PLC2_RANGE_7_1 3325.07 BOOL  ; IN RANGE 7 COUNTER 1
PLC2_RANGE_7_2 3326.07 BOOL  ; IN RANGE 7 COUNTER 2
PLC2_RANGE_8_1 3325.08 BOOL  ; IN RANGE 8 COUNTER 1
PLC2_RANGE_8_2 3326.08 BOOL  ; IN RANGE 8 COUNTER 2
PLC2_RANGE_9_1 3325.09 BOOL  ; IN RANGE 9 COUNTER 1
PLC2_RANGE_9_2 3326.09 BOOL  ; IN RANGE 9 COUNTER 2
PLC3_RANGE_12_1 3325.12 BOOL  ; IN RANGE 12 COUNTER 1
PLC3_RANGE_14_1 3325.14 BOOL  ; IN RANGE 14 COUNTER 1
PRESET_INC_HAG W225.05 BOOL  ; PRESET INCLINOMETER AT HAGENBUCH SYSTEM
PULSE_ENTANCE_GATE_RIGHT W161.00 BOOL  ; PULSE TO OPEN AND CLOSE ENTRANCE GATE RIGHT
PULSE_ENTRANCE_GATE_LEFT W161.01 BOOL  ; PULSE TO OPEN AND CLOSE ENTRANCE GATE LEFT
PULSE_EXIT_GATE W166.00 BOOL  ; PULSE TO OPEN AND CLOSE EXIT GATE
R2_COUNTER4_H 364 INT  ; VALUE COUNTER 4 HIGH WORD
R2_COUNTER_4_L 363 INT  ; VALUE COUNTER 4 LOW WORD
R2_COUNTER_5 369 INT  ; ANALOGE SPANNING KUNSTMATIGE HORIZON
RAMP_DN_X1 D7014 REAL  ; BEGINNING OF RAMP AREA
RAMP_DN_X2 D7016 REAL  ; END OF RAMP AREA
RAMP_DN_Y1 D7010 REAL  ; MAX SPEED AT THE END OF RAMP
RAMP_DN_Y2 D7012 REAL  ; MAX SPEED AT THE BEGINNING OF RAMP
RAMP_FACTOR D182 CHANNEL  ; RAMP FACTOR FOR ARM MOTION
RAMP_UP_X1 D7004 REAL  ; BEGINNING OF RAMP AREA
RAMP_UP_X2 D7006 REAL  ; END OF RAMP AREA
RAMP_UP_Y1 D7000 REAL  ; MAX SPEED AT THE END OF RAMP
RAMP_UP_Y2 D7002 REAL  ; MAX SPEED AT THE BEGINNING OF RAMP
RESULT_A_DN D7074 REAL  ; RESULT A DOWN
RESULT_A_UP D7054 REAL  ; RESULT A UP
RESULT_A_X_DN D7072 REAL  ; RESULT A X DOWN
RESULT_A_X_UP D7052 REAL  ; RESULT A X UP
RESULT_A_Y_DN D7070 REAL  ; RESULT A Y DOWN
RESULT_A_Y_UP D7050 REAL  ; RESULT A Y UP
RESULT_B1_DN D7076 REAL  ; RESULT B1 DOWN
RESULT_B1_UP D7056 REAL  ; RESULT B1 UP
RESULT_B2_DN D7082 REAL  ; RESULT B2 DOWN
RESULT_B2_UP D7062 REAL  ; RESULT B2 UP
RESULT_B_DN D7078 REAL  ; RESULT B DOWN
RESULT_B_UP D7058 REAL  ; RESULT B UP
RESULT_COUNTER_01 2022 INT  ; PULS GETAL ENCODER 1
RESULT_COUNTER_02 2024 INT  ; PULS GETAL ENCODER 2
RESULT_POSITION_VAR_A_DN D7080 REAL  ; RESULT POSITION * VAR A DOWN
RESULT_POSITION_VAR_A_UP D7060 REAL  ; RESULT POSITION * VAR A UP
RES_14_03 14.03 BOOL
RES_14_04 14.04 BOOL
RES_14_05 14.05 BOOL
RES_14_06 14.06 BOOL
RES_14_07 14.07 BOOL
RES_14_08 14.08 BOOL
RES_14_09 14.09 BOOL
RES_14_10 14.10 BOOL
RES_14_11 14.11 BOOL
RES_14_12 14.12 BOOL
RES_14_13 14.13 BOOL
RES_14_14 14.14 BOOL
RES_14_15 14.15 BOOL
STOP_ARM_GOING_UP 3338.00 BOOL  ; STOP ARM GOING UP (LINK BIT TO PLC 1)
TIMER_1 T0001 BOOL L  ; TEST 1
TIMER_2 T0002 BOOL L  ; TEST 2
TIMER_ENC1_FAULT 0150 NUMBER  ; TIMER ENCODER 1 FAUT
TIMER_ENC2_FAULT 0151 NUMBER  ; TIMER ENCODER 2 FAULT
TIMER_PULSE_GATE 0165 NUMBER  ; TIMER FOR OPEN AND CLOSE PULSE EXIT GATE
TIMER_PULSE_GATE_LEFT 0161 NUMBER  ; TIMER FOR OPEN AND CLOSE PULSE ENTRANCE GATE LEFT
TIMER_PULSE_GATE_RIGHT 0160 NUMBER  ; TIMER FOR OPEN AND CLOSE PULSE ENTRANCE GATE RIGHT
TIMER_RESET_BIT 0301 NUMBER  ; TIMER RESET STOP ARM GOING UP BIT
TIMER_STOP_ARM_UP 0300 NUMBER  ; TIMER STOP ARM UP
T_ALARM_1_0161_SET T0021 BOOL
T_ALARM_1_0162_SET T0022 BOOL
T_ALARM_1_0164_SET T0023 BOOL
T_ALARM_1_1191 0320 NUMBER  ; Timer Alarm 1191
T_ALARM_1_1192 0321 NUMBER  ; Timer Alarm 1192
T_ALARM_1_1347 T0205 BOOL
T_ALARM_1_1347_SET 205 NUMBER
T_ALARM_1_1350 T0206 BOOL
T_ALARM_1_1350_SET 206 NUMBER
T_ALARM_1_1453 T0223 BOOL  ; ALARM 1-1453 SIGNAL STATUS VALVE 47 NOT OK
T_ALARM_1_1456 0223 NUMBER  ; ALARM 1-1456 INFO LINK HAGENBUCH (FIBRE OPTIK) NOT AVAILABLE
T_ALARM_1_1457 0224 NUMBER  ; ALARM 1-1457 INFO LINK HAGENBUCH TOO MANY ERRORS
T_ALARM_1_1458 0225 NUMBER  ; ALARM 1-1458 INCLINOMETER TO STABILIZE THE ISLAND NOT OK
T_ALARM_1_1459 0226 NUMBER  ; ALARM 1-1459 STABLIZATION ANGLE ERROR (NORMAL BEFORE TILT SWITCH ERROR)
T_ALARM_1_1460 0227 NUMBER  ; ALARM 1-1460 STABLIZATION PUMP OUT OF ZERO POSITION (MUST BE ZERO POSITION WHEN INLAND IN HOME POSITION)
T_ALARM_1_1461 0228 NUMBER  ; ALARM 1-1461 STABLIZATION PUMP NOT OK
T_ALARM_1_1462_OFF 0231 NUMBER  ; ALARM 1-1462 HARDWARE WATCHDOG FROM HAGENBUCH MISSING TIMER OFF
T_ALARM_1_1462_ON 0230 NUMBER  ; ALARM 1-1462 HARDWARE WATCHDOG FROM HAGENBUCH MISSING TIMER ON
T_ARM_HYDRAULIC_ON 0240 NUMBER  ; TIMER ARM HYDRAULIC ON
T_EILAND_BOVEN T0115 BOOL  ; EILAND TIJD BOVEN
T_Hydr_Main_Pump_Arm_On 0194 NUMBER  ; Hydraulic main pump arm on delay timer
T_ING_L_DICHT T0163 BOOL  ; Max Tijd Sluit Linker Poortjes Oever
T_ING_L_DICHT_SET 161 NUMBER  ; MAX TIJD SLUITEN INGANGS POORT LINKS
T_ING_L_OPEN T0162 BOOL  ; Max Tijd Open Linker Poortjes Oever
T_ING_L_OPEN_SET 160 NUMBER  ; MAX TIJD OPENE INGANG LINKS
T_ING_R_DICHT T0161 BOOL  ; Max Tijd Sluit Rechter Poortjes Oever
T_ING_R_DICHT_SET 163 NUMBER  ; MAX TIJD OPEPEN INGANGS POORTEN RECHTS
T_ING_R_OPEN T0160 BOOL  ; Max Tijd Open Rechter Poortjes Oever
T_ING_R_OPEN_SET 162 NUMBER  ; MAX TIJD OPEPEN INGANGS POORT RECTS
T_ISLAND_HYDRAULIC_ON 0241 NUMBER  ; TIMER ISLAND HYDRAULIC ON
T_Input_0_00 500 NUMBER
T_MS_11Q08_not_OK 0195 NUMBER  ; Hydraulic main pump arm MS 11Q08 not OK
T_MS_11Q10_not_OK 0196 NUMBER  ; Hydraulic main pump arm MS 11Q10 not OK
T_MS_11Q12_not_OK 0197 NUMBER  ; Hydraulic main pump arm MS 11Q12 not OK
T_Open_Uitgangs_poortjes T0165 BOOL  ; Maximale tijd Open Uitgangs Poortjes
T_PRESET_INC_HAGENBUCH 0311 NUMBER  ; PRESET INCLINOMETER HAGENBUCH
T_RESET_HAGENBUCH 0310 NUMBER  ; TIMER RESET ERROR HAGENBUCH SYSTEM
T_SNELHEID 145 NUMBER  ; SNELHEIDS METING ARM
T_SNELHEID_ACT T0145 BOOL  ; TIMER TBV ARM SNELEHEID
T_STUURDRUK_SET_GROND 170 NUMBER  ; DELAY STUURDRUK AANWEZIG
T_STUUR_DRUK T0170 BOOL  ; DELAY STUURDRUK MOET AANWEZIG ZIJN
T_STUUR_DRUK_EIL T0220 BOOL  ; STUURDRUK AANWEZIG EILAND
T_SUURDRUK_EILAND_SET 220 NUMBER  ; DELAY STUUR DRUK AANWEZIG
T_UITG_DICHT T0169 BOOL  ; MAX TIJD UITGANGS POORT SLUITEN
T_UITG_DICHT_SET 169 NUMBER  ; MAX TIJD SLUITEN UITGANGS POORT
T_UITG_OPEN T0165 BOOL  ; MAX TIJD OPENEN UITGANGS POORT
T_UITG_OPEN_SET 165 NUMBER  ; MAX TIJD OPENEN UITGANGS POORTEN
T_Watchdog_Pulse_Check_Plc_2_H T0020 BOOL
T_Watchdog_Pulse_Check_Plc_2_L T0024 BOOL
T_Watchdog_Pulse_Check_Plc_2_Set_H 20 NUMBER
T_Watchdog_Pulse_Check_Plc_2_Set_L 25 NUMBER
T_eilandpoort_set 164 NUMBER  ; delay eilandpoort melding
T_eilandpoortje_act T0164 BOOL  ; delay eiland poort melding
Test_Speed D7500 REAL
U2_72K10 60.03 BOOL  ; ENABLE LINKSOM FREQ.REGELAAR MOTOREN ROTATIE
U2_72K12 60.04 BOOL  ; VRIJGEVEN MOTORREM 1,2,3 EN 4 ROTATIE EILAND
U2_72K14 60.05 BOOL  ; BYPASS ISLAND STABILISATION PUMP
U2_72K16 60.06 BOOL  ; VRIJGAVE POORTJES EILAND
U2_72K18 60.07 BOOL  ; BYPASS ISLAND STABILISATION CYLINDER
U2_72K6 60.01 BOOL L  ; VOEDING FREQ.REGELAAR MOTOREN ROTATIE
U2_72K8 60.02 BOOL  ; ENABLE RECHTSOM FREQ.REGELAAR MOTOREN ROTATIE
U2_73K6 61.02 BOOL  ; HOOFDMOTOR HYDRAULIEK EILAND
U2_73K8 61.03 BOOL  ; VRIJGAVE POORTJES EILAND
U2_73Q4 61.01 BOOL  ; STUURPOMP HYDRAULIEK EILAND
U2_CNT4_COUNT_READ 64.06 BOOL  ; READ COUNTER VALUE
U2_CNT4_COUNT_SET 64.02 BOOL  ; COUNTING SET BIT
U2_CNT4_MODE_1 64.11 BOOL  ; DIFF PHASE 1x
U2_CNT4_MODE_2 64.10 BOOL  ; DIFF PHASE 1x
U2_CNT4_MODE_3 64.12 BOOL  ; RESET MODE
U2_CNT4_MODE_4 64.13 BOOL  ; RESET MODE
U2_CNT4_MODE_5 64.14 BOOL  ; RESET MODE
U2_CNT4_MODE_7 64.03 BOOL  ; DATA MODE 0=BCD 1=HEX
U2_CNT4_RESET 64.07 BOOL  ; INTERNAL RESET
U2_NOOD_PCL1A 60.00 BOOL L  ; NOODSTOP CIRCUIT REMOTE I/O PLC1
U2_NOOD_PCL1B 61.00 BOOL  ; NOODSTOP CIRCUIT REMOTE I/O PLC1
U2_RES_01 61.07 BOOL
U2_SHOWLIGHT_01 61.05 BOOL  ; SHOWLIGHT 01
U2_SHOWLIGHT_02 61.06 BOOL  ; SHOWLIGHT 02
UPS_fault H121.03 BOOL  ; UPS in storing of batterij bedrijf
U_44SH12 13.14 BOOL  ; Ingangs poortjes links oever
U_44SH14 13.15 BOOL  ; Ingangs Poortjes Rechts Oever
U_55K4 8.01 BOOL  ; WATCH DOG PLC 1 (UITGANG DEFECT!!!)
U_85K10 8.04 BOOL  ; ONTGRENDELEN TOURNIQUET LINKS
U_85K12 8.05 BOOL  ; ONTGRENDELEN TOURNIQUET RECHTS
U_85K4 8.07 BOOL  ; Tijdelijke uitgang tbv watchdog
U_85K4_1 7.00 BOOL  ; WATCH DOG PLC 2 NIEUW
U_85Y14 8.06 BOOL  ; POORTJE RECHTS INGANG OPENEN (OEVER)
U_85Y6 8.02 BOOL  ; ARM OMHOOG KLEP 1
U_85Y8 8.03 BOOL  ; ARM OMLAAG KLEP 1
U_86Y10 9.04 BOOL  ; ARM OMLAAG KLEP 3
U_86Y4 9.01 BOOL  ; ARM OMHOOG KLEP 2
U_86Y6 9.02 BOOL  ; ARM OMLAAG KLEP 2
U_86Y8 9.03 BOOL  ; ARM OMHOOG KLEP 3
U_87K8 10.03 BOOL  ; START HOOFDMOTOR HYDRAULIEK UNIT ARM
U_87Q10 10.04 BOOL  ; START STUURPOMP HYDRAULIEK UNIT ARM
U_87Q12 10.05 BOOL  ; START SMEERTOESTEL HYDRAULIEK UNIT ARM
U_87Q14 10.06 BOOL  ; START OLIEREINIGING HYDRAULIEK UNIT ARM
U_87Q6 10.02 BOOL  ; START OLIEKOELER HYDRAULIEK UNIT ARM
U_87Y2 10.00 BOOL  ; POORTJE UITGANG OPENEN (OEVER)
U_87Y4 10.01 BOOL  ; POORTJE UITGANG SLUITEN (OEVER)
U_88Z12 11.05 BOOL  ; ALGEMEEN ALARM ZOEMER
U_91H10 13.04 BOOL  ; ALGEMEEN ALARM
U_91H12 13.05 BOOL  ; KLAAR VOOR SHOW
U_91H14 13.06 BOOL  ; TOURNIQUET LINKS ONTGRENDELD
U_91H16 13.07 BOOL  ; TOURNIQUET RECHTS ONTGRENDELD
U_91H18 13.08 BOOL  ; ARM (EILAND) OMHOOG
U_91H2 13.00 BOOL  ; STUURSPANNING IN
U_91H4 13.01 BOOL  ; HAND BEDRIJF
U_91H6 13.02 BOOL  ; AUTOMATISCH BEDRIJF
U_91H8 13.03 BOOL  ; POMPEN IN BEDRIJF
U_92H12 13.13 BOOL  ; Reset Noodstop
U_92H2 13.09 BOOL  ; ARM (EILAND) OMLAAG
U_92H4 13.10 BOOL  ; EILAND ROTATIE LINKSOM
U_92H6 13.11 BOOL  ; EILAND ROTATIE RECHTSOM
U_92H8 13.12 BOOL  ; Service mode
U_ANA_ARM 2041 CHANNEL  ; ANALOOG _UIT_CHAN1 TBV ARM BESTURING
U_Analog_Uit_Ch2 66 CHANNEL  ; ANALOG OUTPUT ARM POSITION IN DEGREE
U_Analog_Uit_Ch4 68 CHANNEL  ; ANALOG OUTPUT ARM SPEED IN DEGREE/MINUTE
U_ENAB_ANA_CHAN1 2040.00 BOOL  ; CHAN 1 ENABLE
U_ENTRACE_GATE_RIGHT 14.00 BOOL  ; ENTRANCE GATE RIGHT
U_ENTRANCE_GATE_LEFT 14.01 BOOL  ; ENTRANCE GATE LEFT
U_EXIT_GATE 14.02 BOOL  ; EXIT GATE
U_HAG_BIT_10 61.04 BOOL  ; HAGENBUCH TILT SENSOREN OK
U_HAG_PRESET 9.05 BOOL  ; HAGENBUCH PRESET INCLINOMETER
U_HAG_RESET 9.06 BOOL  ; HAGENBUCH ALARM RESET
U_Ingangs_Poortje_Links_Oever 12.04 BOOL
U_Ingangs_Poortje_Rechts_Oever 12.00 BOOL
U_NS_PLC1A 8.00 BOOL  ; NOODSTOP CIRCUIT PLC 1
U_NS_PLC1B 9.00 BOOL  ; NOODSTOP CIRCUIT PLC 1
U_Open_Ingangs_Poortje_2_Links_Oever 12.05 BOOL
U_Open_Ingangs_Poortje_2_Rechts_Oever 12.01 BOOL  ; Open Ingangs Poortje 2 Rechter zijde Oever
U_Open_Uitgangs_Poortje_2_Oever 12.09 BOOL
U_RES_10_07 10.07 BOOL  ; RESERVE
U_Res_noodstop 9.07 BOOL  ; Mogelijk om noodstop te resetten
U_Sluit_Ingangs_Poortje_1_Links_Oever 12.06 BOOL
U_Sluit_Ingangs_Poortje_1_Rechts_Oever 12.02 BOOL  ; Sluit Poortje 1 Rechter zijde Oever
U_Sluit_Ingangs_Poortje_2_Links_Oever 12.07 BOOL
U_Sluit_Ingangs_Poortje_2_Rechts_Oever 12.03 BOOL  ; Sluit Poortje 2 Rechter zijde Oever
U_Sluit_Uitgangs_Poortje_1_Oever 12.10 BOOL
U_Sluit_Uitgangs_Poortje_2_Oever 12.11 BOOL
U_Uitgangs_Poortje_Oever 12.08 BOOL
W_ING_PRT_EIL_GESL W210.05 BOOL  ; Ingangs Poortjes Eiland Gesloten Plc 1 & 2 & 3
W_RANGE0_CNT1 W125.00 BOOL  ; ARM IN RANGE 0
W_RANGE0_CNT2 W126.00 BOOL  ; ARM IN RANGE 0
W_RANGE0_PLC1 3036.00 BOOL  ; ARM IN RANGE 0
W_RANGE0_PLC2 3336.00 BOOL  ; ARM IN RANGE 0
W_RANGE10_CNT1 W125.10 BOOL  ; ARM IN RANGE 10
W_RANGE10_CNT2 W126.10 BOOL  ; ARM IN RANGE 10
W_RANGE10_PLC1 3036.10 BOOL  ; ARM IN RANGE 10
W_RANGE10_PLC2 3336.10 BOOL  ; ARM IN RANGE 10
W_RANGE11_CNT1 W125.11 BOOL  ; ARM IN RANGE 11
W_RANGE11_CNT2 W126.11 BOOL  ; ARM IN RANGE 11
W_RANGE11_PLC1 3036.11 BOOL  ; ARM IN RANGE 11
W_RANGE11_PLC2 3336.11 BOOL  ; ARM IN RANGE 11
W_RANGE12_CNT1 W125.12 BOOL  ; ARM IN RANGE 12
W_RANGE12_CNT2 W126.12 BOOL  ; ARM IN RANGE 12
W_RANGE12_PLC1 3036.12 BOOL  ; ARM IN RANGE 12
W_RANGE12_PLC2 3336.12 BOOL  ; ARM IN RANGE 12
W_RANGE13_CNT1 W125.13 BOOL  ; ARM IN RANGE 13
W_RANGE13_CNT2 W126.13 BOOL  ; ARM IN RANGE 13
W_RANGE13_PLC1 3036.13 BOOL  ; ARM IN RANGE 13
W_RANGE13_PLC2 3336.13 BOOL  ; ARM IN RANGE 13
W_RANGE14_CNT1 W125.14 BOOL  ; ARM IN RANGE 14
W_RANGE14_CNT2 W126.14 BOOL  ; ARM IN RANGE 14
W_RANGE14_PLC1 3036.14 BOOL  ; ARM IN RANGE 14
W_RANGE14_PLC2 3336.14 BOOL  ; ARM IN RANGE 14
W_RANGE15_CNT1 W125.15 BOOL  ; ARM IN RANGE 15
W_RANGE15_CNT2 W126.15 BOOL  ; ARM IN RANGE 15
W_RANGE15_PLC1 3036.15 BOOL  ; ARM IN RANGE 15
W_RANGE15_PLC2 3336.15 BOOL  ; ARM IN RANGE 15
W_RANGE1_CNT1 W125.01 BOOL  ; ARM IN RANGE 1
W_RANGE1_CNT2 W126.01 BOOL  ; ARM IN RANGE 1
W_RANGE1_PLC1 3036.01 BOOL  ; ARM IN RANGE 1
W_RANGE1_PLC2 3336.01 BOOL  ; ARM IN RANGE 1
W_RANGE2_CNT1 W125.02 BOOL  ; ARM IN RANGE 2
W_RANGE2_CNT2 W126.02 BOOL  ; ARM IN RANGE 2
W_RANGE2_PLC1 3036.02 BOOL  ; ARM IN RANGE 2
W_RANGE2_PLC2 3336.02 BOOL  ; ARM IN RANGE 2
W_RANGE3_CNT1 W125.03 BOOL  ; ARM IN RANGE 3
W_RANGE3_CNT2 W126.03 BOOL  ; ARM IN RANGE 3
W_RANGE3_PLC1 3036.03 BOOL  ; ARM IN RANGE 3
W_RANGE3_PLC2 3336.03 BOOL  ; ARM IN RANGE 3
W_RANGE4_CNT1 W125.04 BOOL  ; ARM IN RANGE 4
W_RANGE4_CNT2 W126.04 BOOL  ; ARM IN RANGE 4
W_RANGE4_PLC1 3036.04 BOOL  ; ARM IN RANGE 4
W_RANGE4_PLC2 3336.04 BOOL  ; ARM IN RANGE 4
W_RANGE5_CNT1 W125.05 BOOL  ; ARM IN RANGE 5
W_RANGE5_CNT2 W126.05 BOOL  ; ARM IN RANGE 5
W_RANGE5_PLC1 3036.05 BOOL  ; ARM IN RANGE 5
W_RANGE5_PLC2 3336.05 BOOL  ; ARM IN RANGE 5
W_RANGE6_CNT1 W125.06 BOOL  ; ARM IN RANGE 6
W_RANGE6_CNT2 W126.06 BOOL  ; ARM IN RANGE 6
W_RANGE6_PLC1 3036.06 BOOL  ; ARM IN RANGE 6
W_RANGE6_PLC2 3336.06 BOOL  ; ARM IN RANGE 6
W_RANGE7_CNT1 W125.07 BOOL  ; ARM IN RANGE 7
W_RANGE7_CNT2 W126.07 BOOL  ; ARM IN RANGE 7
W_RANGE7_PLC1 3036.07 BOOL  ; ARM IN RANGE 7
W_RANGE7_PLC2 3336.07 BOOL  ; ARM IN RANGE 7
W_RANGE8_CNT1 W125.08 BOOL  ; ARM IN RANGE 8
W_RANGE8_CNT2 W126.08 BOOL  ; ARM IN RANGE 8
W_RANGE8_PLC1 3036.08 BOOL  ; ARM IN RANGE 8
W_RANGE8_PLC2 3336.08 BOOL  ; ARM IN RANGE 8
W_RANGE9_CNT1 W125.09 BOOL  ; ARM IN RANGE 9
W_RANGE9_CNT2 W126.09 BOOL  ; ARM IN RANGE 9
W_RANGE9_PLC1 3036.09 BOOL  ; ARM IN RANGE 9
W_RANGE9_PLC2 3336.09 BOOL  ; ARM IN RANGE 9
com1_Eiland_Home 3024.02 BOOL  ; Het Eiland Is geheel Links- of Rechtsom Gedraaid
t_diff_arm T0175 BOOL  ; verschil soll-ist arm
t_diff_soll_arm 175 NUMBER  ; diff soll ist verschil arm
t_eiland_boven 0115 NUMBER  ; eiland boven tijd

## Program ALGEMEEN (cyclic task 0)
Local symbols
M_ALARM_1_0000 H100.00 BOOL  ; Alarm 1 - 0000 Er is minstens 1 Alarm in de File Main (Alarmen 1 - 0000 t/m 1 -  0031)
M_ALARM_1_0032 H102.00 BOOL  ; Alarm 1 - 0032 Er is minstens 1 Alarm in de Controllink (Alarmen 1 - 0032 t/m 1 -  0063)
M_ALARM_1_0096 H106.00 BOOL  ; Alarm 1 - 0096 Er is minstens 1 Alarm in de Data-Opslag (Alarmen 1 - 0096 t/m 1 -  0127)
M_ALARM_1_0128 H108.00 BOOL  ; Alarm 1-0128 Er is minstens 1 alarm in de I/O Controle afhandeling
M_Alarm_H100_H108 W36.00 BOOL
M_Alarm_H110_H118 W36.01 BOOL
M_Alarm_H120_H128 W36.02 BOOL
M_Alarm_H130_H138 W36.03 BOOL
M_Alarm_H140_H148 W36.04 BOOL
M_Alarm_H150_H158 W36.05 BOOL
M_Alarm_H160_H168 W36.06 BOOL
M_Alarm_H170_H178 W36.07 BOOL
M_Alarm_H180_H188 W36.08 BOOL
M_Alarm_H190_H198 W36.09 BOOL
U_WCD_1 11.06 BOOL
U_WCD_2 11.07 BOOL
U_WCD_5 61.07 BOOL

### Section Main

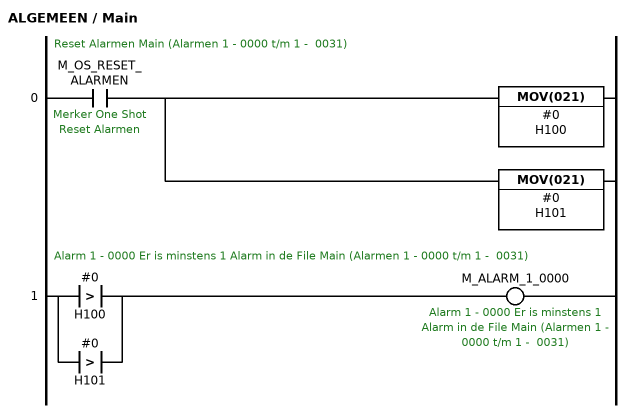
; rung 0: Reset Alarmen Main (Alarmen 1 - 0000 t/m 1 -  0031)
LD M_OS_RESET_ALARMEN  ; Merker One Shot Reset Alarmen
MOV(021) #0 H100
MOV(021) #0 H101
; rung 1: Alarm 1 - 0000 Er is minstens 1 Alarm in de File Main (Alarmen 1 - 0000 t/m 1 -  0031)
LD>(320) #0 H100
OR>(320) #0 H101
OUT M_ALARM_1_0000  ; Alarm 1 - 0000 Er is minstens 1 Alarm in de File Main (Alarmen 1 - 0000 t/m 1 -  0031)

### Section Control_Link

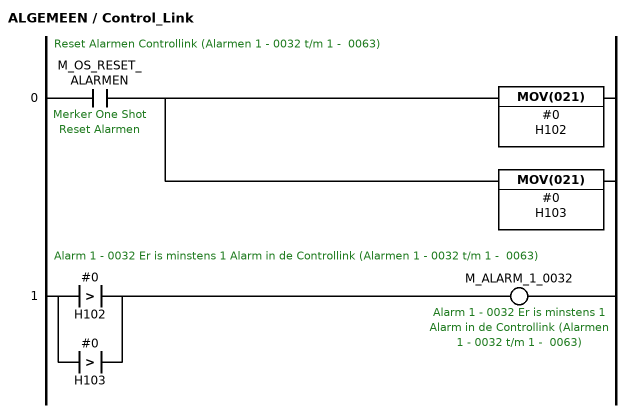
; rung 0: Reset Alarmen Controllink (Alarmen 1 - 0032 t/m 1 -  0063)
LD M_OS_RESET_ALARMEN  ; Merker One Shot Reset Alarmen
MOV(021) #0 H102
MOV(021) #0 H103
; rung 1: Alarm 1 - 0032 Er is minstens 1 Alarm in de Controllink (Alarmen 1 - 0032 t/m 1 -  0063)
LD>(320) #0 H102
OR>(320) #0 H103
OUT M_ALARM_1_0032  ; Alarm 1 - 0032 Er is minstens 1 Alarm in de Controllink (Alarmen 1 - 0032 t/m 1 -  0063)

### Section Device_net

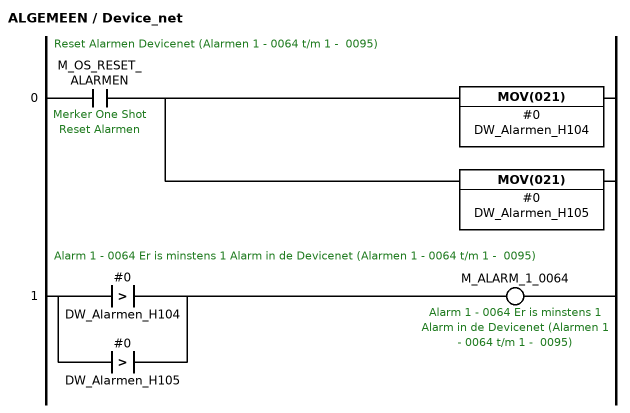
; rung 0: Reset Alarmen Devicenet (Alarmen 1 - 0064 t/m 1 -  0095)
LD M_OS_RESET_ALARMEN  ; Merker One Shot Reset Alarmen
MOV(021) #0 DW_Alarmen_H104
MOV(021) #0 DW_Alarmen_H105
; rung 1: Alarm 1 - 0064 Er is minstens 1 Alarm in de Devicenet (Alarmen 1 - 0064 t/m 1 -  0095)
LD>(320) #0 DW_Alarmen_H104
OR>(320) #0 DW_Alarmen_H105
OUT M_ALARM_1_0064  ; Alarm 1 - 0064 Er is minstens 1 Alarm in de Devicenet (Alarmen 1 - 0064 t/m 1 -  0095)

### Section Data_Opslag

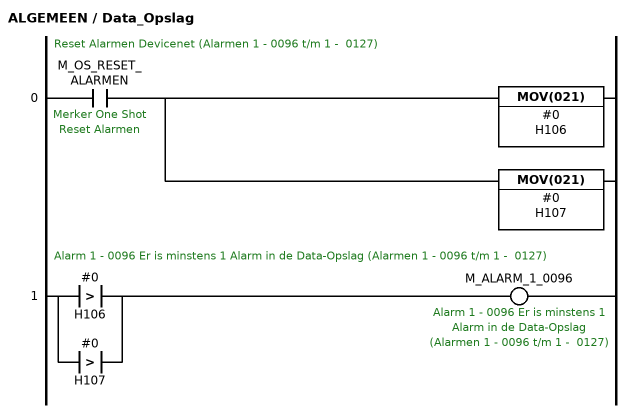
; rung 0: Reset Alarmen Devicenet (Alarmen 1 - 0096 t/m 1 -  0127)
LD M_OS_RESET_ALARMEN  ; Merker One Shot Reset Alarmen
MOV(021) #0 H106
MOV(021) #0 H107
; rung 1: Alarm 1 - 0096 Er is minstens 1 Alarm in de Data-Opslag (Alarmen 1 - 0096 t/m 1 -  0127)
LD>(320) #0 H106
OR>(320) #0 H107
OUT M_ALARM_1_0096  ; Alarm 1 - 0096 Er is minstens 1 Alarm in de Data-Opslag (Alarmen 1 - 0096 t/m 1 -  0127)

### Section I_O_Controle

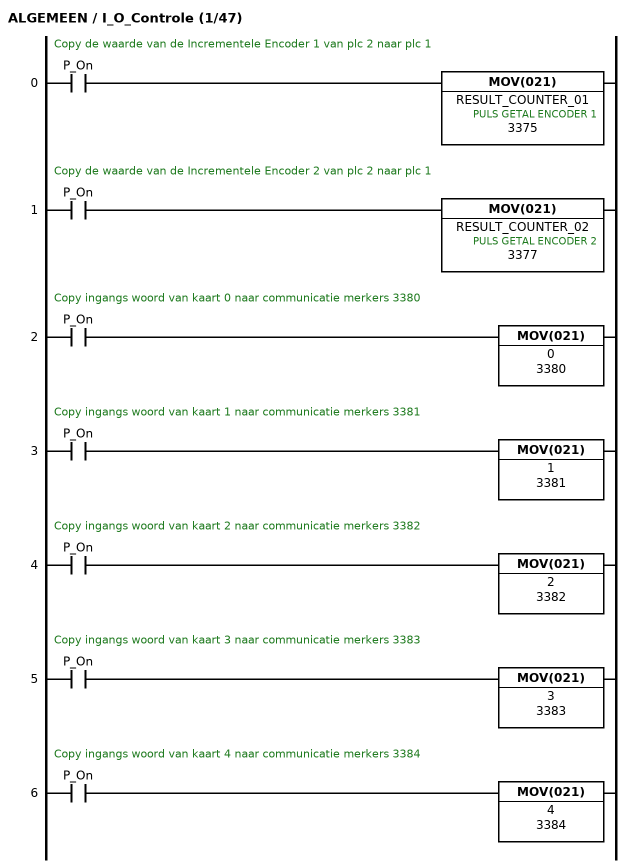
; rung 0: Copy de waarde van de Incrementele Encoder 1 van plc 2 naar plc 1
LD P_On
MOV(021) RESULT_COUNTER_01 3375  ; PULS GETAL ENCODER 1
; rung 1: Copy de waarde van de Incrementele Encoder 2 van plc 2 naar plc 1
LD P_On
MOV(021) RESULT_COUNTER_02 3377  ; PULS GETAL ENCODER 2
; rung 2: Copy ingangs woord van kaart 0 naar communicatie merkers 3380
LD P_On
MOV(021) 0 3380
; rung 3: Copy ingangs woord van kaart 1 naar communicatie merkers 3381
LD P_On
MOV(021) 1 3381
; rung 4: Copy ingangs woord van kaart 2 naar communicatie merkers 3382
LD P_On
MOV(021) 2 3382
; rung 5: Copy ingangs woord van kaart 3 naar communicatie merkers 3383
LD P_On
MOV(021) 3 3383
; rung 6: Copy ingangs woord van kaart 4 naar communicatie merkers 3384
LD P_On
MOV(021) 4 3384

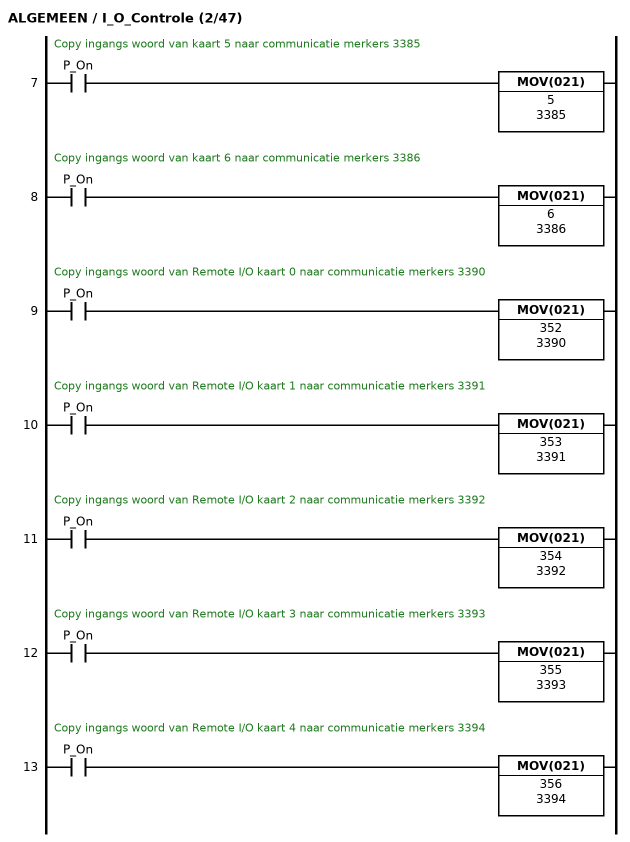
; rung 7: Copy ingangs woord van kaart 5 naar communicatie merkers 3385
LD P_On
MOV(021) 5 3385
; rung 8: Copy ingangs woord van kaart 6 naar communicatie merkers 3386
LD P_On
MOV(021) 6 3386
; rung 9: Copy ingangs woord van Remote I/O kaart 0 naar communicatie merkers 3390
LD P_On
MOV(021) 352 3390
; rung 10: Copy ingangs woord van Remote I/O kaart 1 naar communicatie merkers 3391
LD P_On
MOV(021) 353 3391
; rung 11: Copy ingangs woord van Remote I/O kaart 2 naar communicatie merkers 3392
LD P_On
MOV(021) 354 3392
; rung 12: Copy ingangs woord van Remote I/O kaart 3 naar communicatie merkers 3393
LD P_On
MOV(021) 355 3393
; rung 13: Copy ingangs woord van Remote I/O kaart 4 naar communicatie merkers 3394
LD P_On
MOV(021) 356 3394

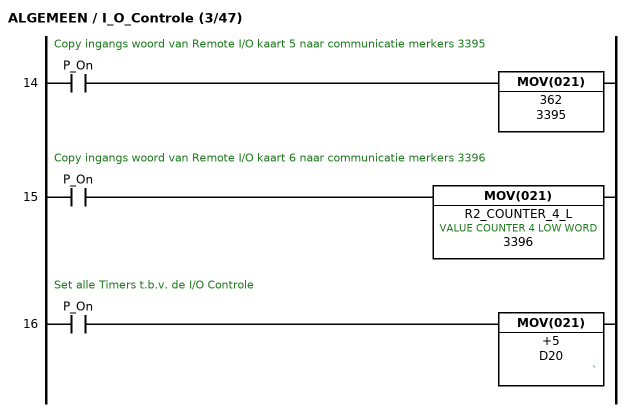
; rung 14: Copy ingangs woord van Remote I/O kaart 5 naar communicatie merkers 3395
LD P_On
MOV(021) 362 3395
; rung 15: Copy ingangs woord van Remote I/O kaart 6 naar communicatie merkers 3396
LD P_On
MOV(021) R2_COUNTER_4_L 3396  ; VALUE COUNTER 4 LOW WORD
; rung 16: Set alle Timers t.b.v. de I/O Controle
LD P_On
MOV(021) +5 D20  ; `

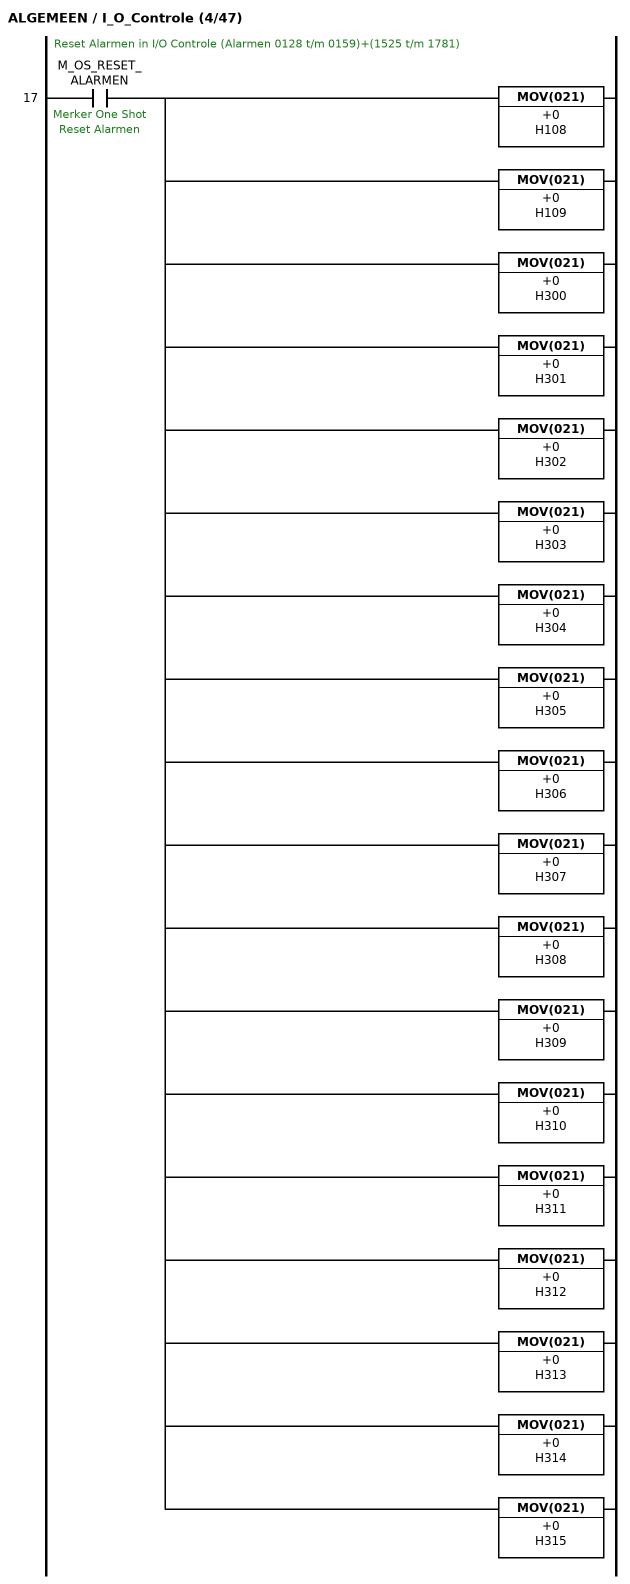
; rung 17: Reset Alarmen in I/O Controle (Alarmen 0128 t/m 0159)+(1525 t/m 1781)
LD M_OS_RESET_ALARMEN  ; Merker One Shot Reset Alarmen
MOV(021) +0 H108
MOV(021) +0 H109
MOV(021) +0 H300
MOV(021) +0 H301
MOV(021) +0 H302
MOV(021) +0 H303
MOV(021) +0 H304
MOV(021) +0 H305
MOV(021) +0 H306
MOV(021) +0 H307
MOV(021) +0 H308
MOV(021) +0 H309
MOV(021) +0 H310
MOV(021) +0 H311
MOV(021) +0 H312
MOV(021) +0 H313
MOV(021) +0 H314
MOV(021) +0 H315

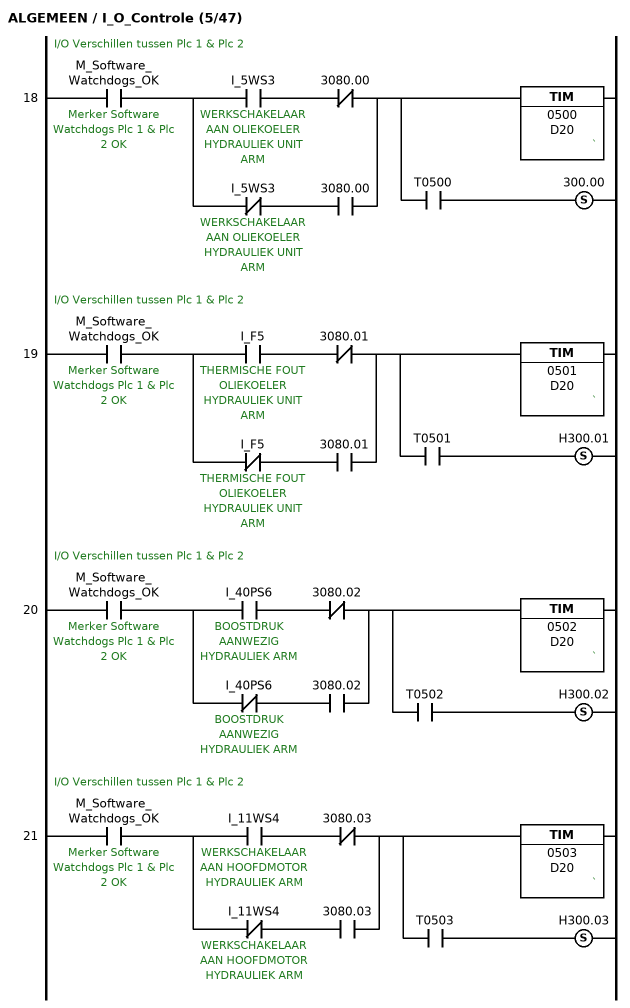
; rung 18: I/O Verschillen tussen Plc 1 & Plc 2
LD M_Software_Watchdogs_OK  ; Merker Software Watchdogs Plc 1 & Plc 2 OK
LD I_5WS3  ; WERKSCHAKELAAR AAN OLIEKOELER HYDRAULIEK UNIT ARM
ANDNOT 3080.00
LDNOT I_5WS3  ; WERKSCHAKELAAR AAN OLIEKOELER HYDRAULIEK UNIT ARM
AND 3080.00
ORLD
ANDLD
TIM 0500 D20  ; `
AND T0500
SET 300.00
; rung 19: I/O Verschillen tussen Plc 1 & Plc 2
LD M_Software_Watchdogs_OK  ; Merker Software Watchdogs Plc 1 & Plc 2 OK
LD I_F5  ; THERMISCHE FOUT OLIEKOELER HYDRAULIEK UNIT ARM
ANDNOT 3080.01
LDNOT I_F5  ; THERMISCHE FOUT OLIEKOELER HYDRAULIEK UNIT ARM
AND 3080.01
ORLD
ANDLD
TIM 0501 D20  ; `
AND T0501
SET H300.01
; rung 20: I/O Verschillen tussen Plc 1 & Plc 2
LD M_Software_Watchdogs_OK  ; Merker Software Watchdogs Plc 1 & Plc 2 OK
LD I_40PS6  ; BOOSTDRUK AANWEZIG HYDRAULIEK ARM
ANDNOT 3080.02
LDNOT I_40PS6  ; BOOSTDRUK AANWEZIG HYDRAULIEK ARM
AND 3080.02
ORLD
ANDLD
TIM 0502 D20  ; `
AND T0502
SET H300.02
; rung 21: I/O Verschillen tussen Plc 1 & Plc 2
LD M_Software_Watchdogs_OK  ; Merker Software Watchdogs Plc 1 & Plc 2 OK
LD I_11WS4  ; WERKSCHAKELAAR AAN HOOFDMOTOR HYDRAULIEK ARM
ANDNOT 3080.03
LDNOT I_11WS4  ; WERKSCHAKELAAR AAN HOOFDMOTOR HYDRAULIEK ARM
AND 3080.03
ORLD
ANDLD
TIM 0503 D20  ; `
AND T0503
SET H300.03

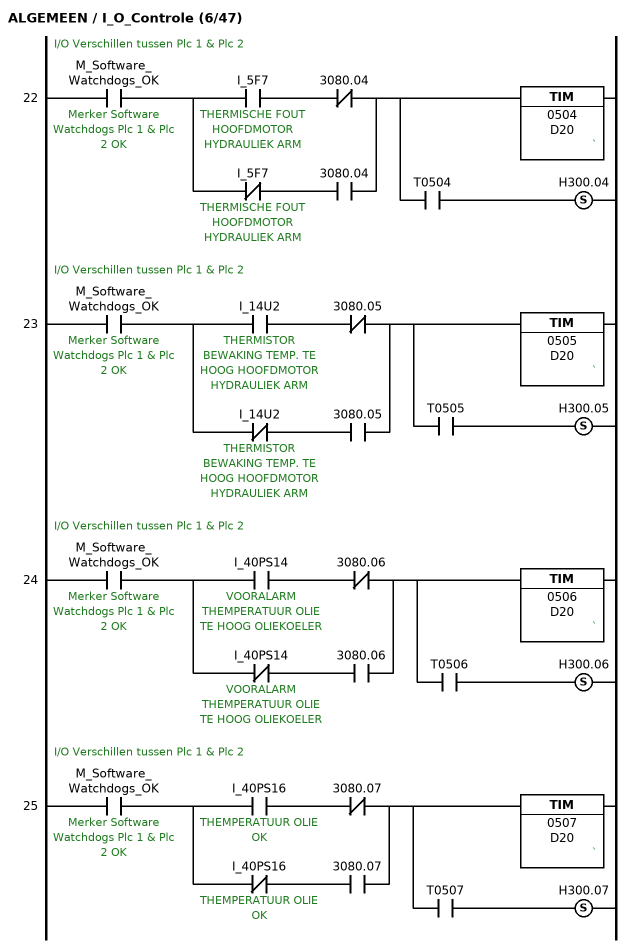
; rung 22: I/O Verschillen tussen Plc 1 & Plc 2
LD M_Software_Watchdogs_OK  ; Merker Software Watchdogs Plc 1 & Plc 2 OK
LD I_5F7  ; THERMISCHE FOUT HOOFDMOTOR HYDRAULIEK ARM
ANDNOT 3080.04
LDNOT I_5F7  ; THERMISCHE FOUT HOOFDMOTOR HYDRAULIEK ARM
AND 3080.04
ORLD
ANDLD
TIM 0504 D20  ; `
AND T0504
SET H300.04
; rung 23: I/O Verschillen tussen Plc 1 & Plc 2
LD M_Software_Watchdogs_OK  ; Merker Software Watchdogs Plc 1 & Plc 2 OK
LD I_14U2  ; THERMISTOR BEWAKING TEMP. TE HOOG HOOFDMOTOR HYDRAULIEK ARM
ANDNOT 3080.05
LDNOT I_14U2  ; THERMISTOR BEWAKING TEMP. TE HOOG HOOFDMOTOR HYDRAULIEK ARM
AND 3080.05
ORLD
ANDLD
TIM 0505 D20  ; `
AND T0505
SET H300.05
; rung 24: I/O Verschillen tussen Plc 1 & Plc 2
LD M_Software_Watchdogs_OK  ; Merker Software Watchdogs Plc 1 & Plc 2 OK
LD I_40PS14  ; VOORALARM THEMPERATUUR OLIE TE HOOG OLIEKOELER
ANDNOT 3080.06
LDNOT I_40PS14  ; VOORALARM THEMPERATUUR OLIE TE HOOG OLIEKOELER
AND 3080.06
ORLD
ANDLD
TIM 0506 D20  ; `
AND T0506
SET H300.06
; rung 25: I/O Verschillen tussen Plc 1 & Plc 2
LD M_Software_Watchdogs_OK  ; Merker Software Watchdogs Plc 1 & Plc 2 OK
LD I_40PS16  ; THEMPERATUUR OLIE OK
ANDNOT 3080.07
LDNOT I_40PS16  ; THEMPERATUUR OLIE OK
AND 3080.07
ORLD
ANDLD
TIM 0507 D20  ; `
AND T0507
SET H300.07

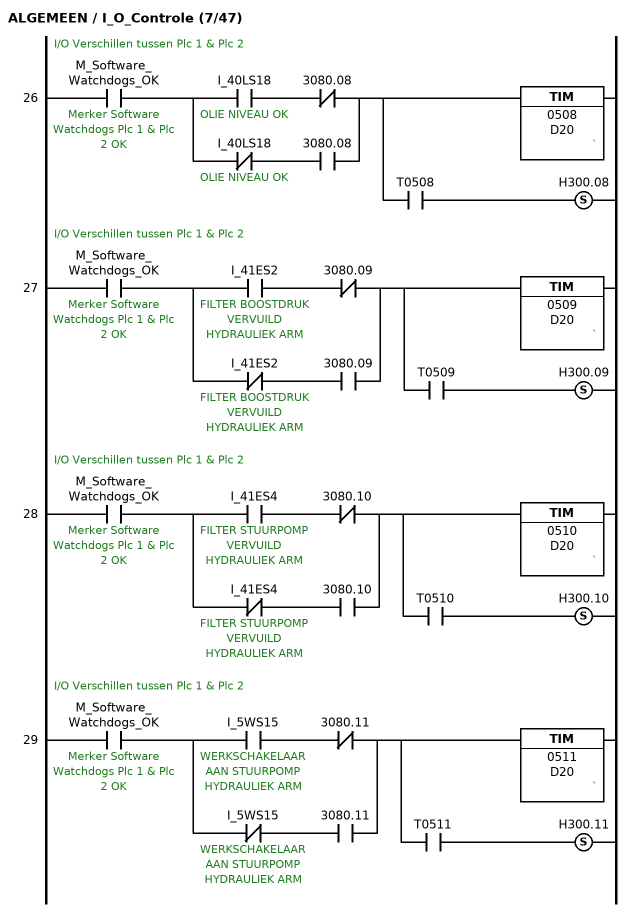
; rung 26: I/O Verschillen tussen Plc 1 & Plc 2
LD M_Software_Watchdogs_OK  ; Merker Software Watchdogs Plc 1 & Plc 2 OK
LD I_40LS18  ; OLIE NIVEAU OK
ANDNOT 3080.08
LDNOT I_40LS18  ; OLIE NIVEAU OK
AND 3080.08
ORLD
ANDLD
TIM 0508 D20  ; `
AND T0508
SET H300.08
; rung 27: I/O Verschillen tussen Plc 1 & Plc 2
LD M_Software_Watchdogs_OK  ; Merker Software Watchdogs Plc 1 & Plc 2 OK
LD I_41ES2  ; FILTER BOOSTDRUK VERVUILD HYDRAULIEK ARM
ANDNOT 3080.09
LDNOT I_41ES2  ; FILTER BOOSTDRUK VERVUILD HYDRAULIEK ARM
AND 3080.09
ORLD
ANDLD
TIM 0509 D20  ; `
AND T0509
SET H300.09
; rung 28: I/O Verschillen tussen Plc 1 & Plc 2
LD M_Software_Watchdogs_OK  ; Merker Software Watchdogs Plc 1 & Plc 2 OK
LD I_41ES4  ; FILTER STUURPOMP VERVUILD HYDRAULIEK ARM
ANDNOT 3080.10
LDNOT I_41ES4  ; FILTER STUURPOMP VERVUILD HYDRAULIEK ARM
AND 3080.10
ORLD
ANDLD
TIM 0510 D20  ; `
AND T0510
SET H300.10
; rung 29: I/O Verschillen tussen Plc 1 & Plc 2
LD M_Software_Watchdogs_OK  ; Merker Software Watchdogs Plc 1 & Plc 2 OK
LD I_5WS15  ; WERKSCHAKELAAR AAN STUURPOMP HYDRAULIEK ARM
ANDNOT 3080.11
LDNOT I_5WS15  ; WERKSCHAKELAAR AAN STUURPOMP HYDRAULIEK ARM
AND 3080.11
ORLD
ANDLD
TIM 0511 D20  ; `
AND T0511
SET H300.11

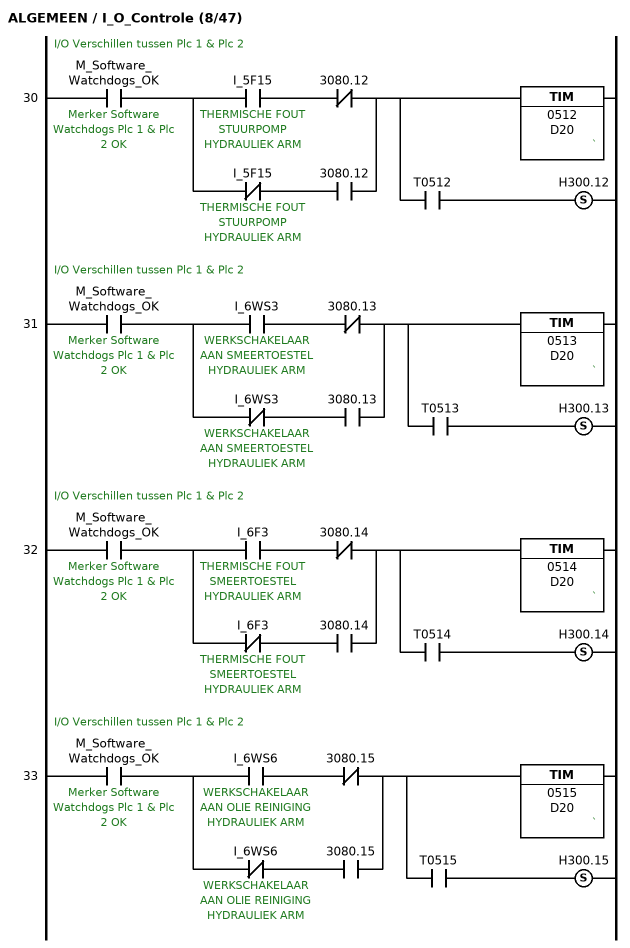
; rung 30: I/O Verschillen tussen Plc 1 & Plc 2
LD M_Software_Watchdogs_OK  ; Merker Software Watchdogs Plc 1 & Plc 2 OK
LD I_5F15  ; THERMISCHE FOUT STUURPOMP HYDRAULIEK ARM
ANDNOT 3080.12
LDNOT I_5F15  ; THERMISCHE FOUT STUURPOMP HYDRAULIEK ARM
AND 3080.12
ORLD
ANDLD
TIM 0512 D20  ; `
AND T0512
SET H300.12
; rung 31: I/O Verschillen tussen Plc 1 & Plc 2
LD M_Software_Watchdogs_OK  ; Merker Software Watchdogs Plc 1 & Plc 2 OK
LD I_6WS3  ; WERKSCHAKELAAR AAN SMEERTOESTEL HYDRAULIEK ARM
ANDNOT 3080.13
LDNOT I_6WS3  ; WERKSCHAKELAAR AAN SMEERTOESTEL HYDRAULIEK ARM
AND 3080.13
ORLD
ANDLD
TIM 0513 D20  ; `
AND T0513
SET H300.13
; rung 32: I/O Verschillen tussen Plc 1 & Plc 2
LD M_Software_Watchdogs_OK  ; Merker Software Watchdogs Plc 1 & Plc 2 OK
LD I_6F3  ; THERMISCHE FOUT SMEERTOESTEL HYDRAULIEK ARM
ANDNOT 3080.14
LDNOT I_6F3  ; THERMISCHE FOUT SMEERTOESTEL HYDRAULIEK ARM
AND 3080.14
ORLD
ANDLD
TIM 0514 D20  ; `
AND T0514
SET H300.14
; rung 33: I/O Verschillen tussen Plc 1 & Plc 2
LD M_Software_Watchdogs_OK  ; Merker Software Watchdogs Plc 1 & Plc 2 OK
LD I_6WS6  ; WERKSCHAKELAAR AAN OLIE REINIGING HYDRAULIEK ARM
ANDNOT 3080.15
LDNOT I_6WS6  ; WERKSCHAKELAAR AAN OLIE REINIGING HYDRAULIEK ARM
AND 3080.15
ORLD
ANDLD
TIM 0515 D20  ; `
AND T0515
SET H300.15

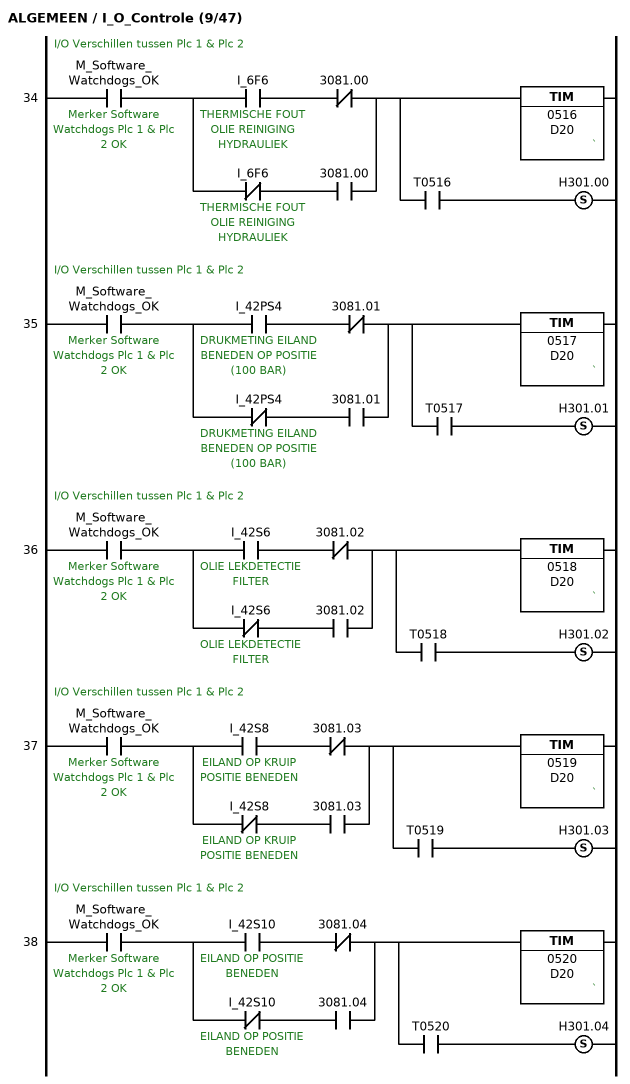
; rung 34: I/O Verschillen tussen Plc 1 & Plc 2
LD M_Software_Watchdogs_OK  ; Merker Software Watchdogs Plc 1 & Plc 2 OK
LD I_6F6  ; THERMISCHE FOUT OLIE REINIGING HYDRAULIEK
ANDNOT 3081.00
LDNOT I_6F6  ; THERMISCHE FOUT OLIE REINIGING HYDRAULIEK
AND 3081.00
ORLD
ANDLD
TIM 0516 D20  ; `
AND T0516
SET H301.00
; rung 35: I/O Verschillen tussen Plc 1 & Plc 2
LD M_Software_Watchdogs_OK  ; Merker Software Watchdogs Plc 1 & Plc 2 OK
LD I_42PS4  ; DRUKMETING EILAND BENEDEN OP POSITIE (100 BAR)
ANDNOT 3081.01
LDNOT I_42PS4  ; DRUKMETING EILAND BENEDEN OP POSITIE (100 BAR)
AND 3081.01
ORLD
ANDLD
TIM 0517 D20  ; `
AND T0517
SET H301.01
; rung 36: I/O Verschillen tussen Plc 1 & Plc 2
LD M_Software_Watchdogs_OK  ; Merker Software Watchdogs Plc 1 & Plc 2 OK
LD I_42S6  ; OLIE LEKDETECTIE FILTER
ANDNOT 3081.02
LDNOT I_42S6  ; OLIE LEKDETECTIE FILTER
AND 3081.02
ORLD
ANDLD
TIM 0518 D20  ; `
AND T0518
SET H301.02
; rung 37: I/O Verschillen tussen Plc 1 & Plc 2
LD M_Software_Watchdogs_OK  ; Merker Software Watchdogs Plc 1 & Plc 2 OK
LD I_42S8  ; EILAND OP KRUIP POSITIE BENEDEN
ANDNOT 3081.03
LDNOT I_42S8  ; EILAND OP KRUIP POSITIE BENEDEN
AND 3081.03
ORLD
ANDLD
TIM 0519 D20  ; `
AND T0519
SET H301.03
; rung 38: I/O Verschillen tussen Plc 1 & Plc 2
LD M_Software_Watchdogs_OK  ; Merker Software Watchdogs Plc 1 & Plc 2 OK
LD I_42S10  ; EILAND OP POSITIE BENEDEN
ANDNOT 3081.04
LDNOT I_42S10  ; EILAND OP POSITIE BENEDEN
AND 3081.04
ORLD
ANDLD
TIM 0520 D20  ; `
AND T0520
SET H301.04

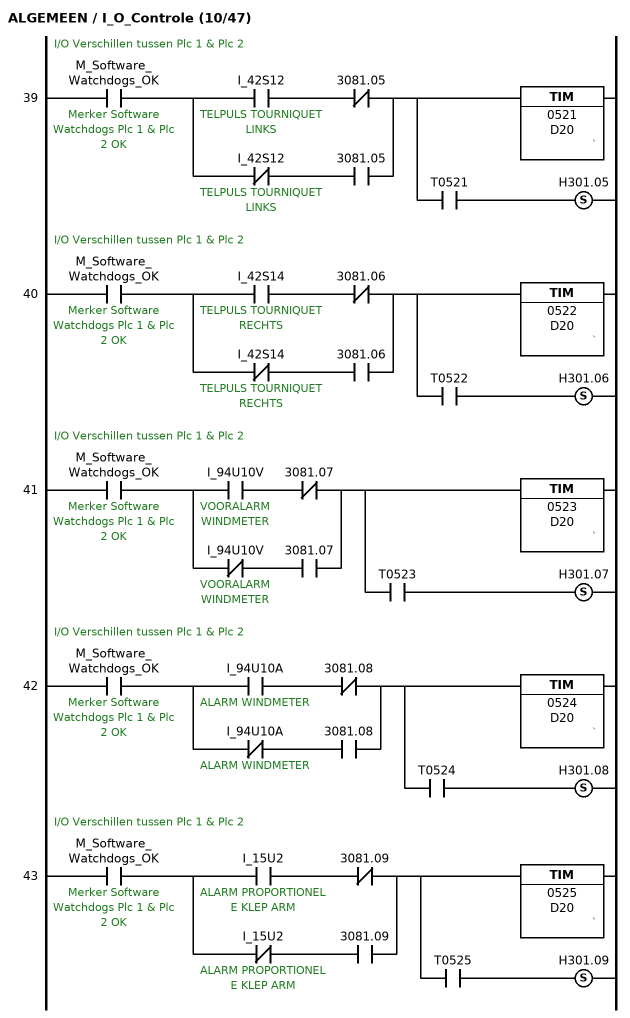
; rung 39: I/O Verschillen tussen Plc 1 & Plc 2
LD M_Software_Watchdogs_OK  ; Merker Software Watchdogs Plc 1 & Plc 2 OK
LD I_42S12  ; TELPULS TOURNIQUET LINKS
ANDNOT 3081.05
LDNOT I_42S12  ; TELPULS TOURNIQUET LINKS
AND 3081.05
ORLD
ANDLD
TIM 0521 D20  ; `
AND T0521
SET H301.05
; rung 40: I/O Verschillen tussen Plc 1 & Plc 2
LD M_Software_Watchdogs_OK  ; Merker Software Watchdogs Plc 1 & Plc 2 OK
LD I_42S14  ; TELPULS TOURNIQUET RECHTS
ANDNOT 3081.06
LDNOT I_42S14  ; TELPULS TOURNIQUET RECHTS
AND 3081.06
ORLD
ANDLD
TIM 0522 D20  ; `
AND T0522
SET H301.06
; rung 41: I/O Verschillen tussen Plc 1 & Plc 2
LD M_Software_Watchdogs_OK  ; Merker Software Watchdogs Plc 1 & Plc 2 OK
LD I_94U10V  ; VOORALARM WINDMETER
ANDNOT 3081.07
LDNOT I_94U10V  ; VOORALARM WINDMETER
AND 3081.07
ORLD
ANDLD
TIM 0523 D20  ; `
AND T0523
SET H301.07
; rung 42: I/O Verschillen tussen Plc 1 & Plc 2
LD M_Software_Watchdogs_OK  ; Merker Software Watchdogs Plc 1 & Plc 2 OK
LD I_94U10A  ; ALARM WINDMETER
ANDNOT 3081.08
LDNOT I_94U10A  ; ALARM WINDMETER
AND 3081.08
ORLD
ANDLD
TIM 0524 D20  ; `
AND T0524
SET H301.08
; rung 43: I/O Verschillen tussen Plc 1 & Plc 2
LD M_Software_Watchdogs_OK  ; Merker Software Watchdogs Plc 1 & Plc 2 OK
LD I_15U2  ; ALARM PROPORTIONELE KLEP ARM
ANDNOT 3081.09
LDNOT I_15U2  ; ALARM PROPORTIONELE KLEP ARM
AND 3081.09
ORLD
ANDLD
TIM 0525 D20  ; `
AND T0525
SET H301.09

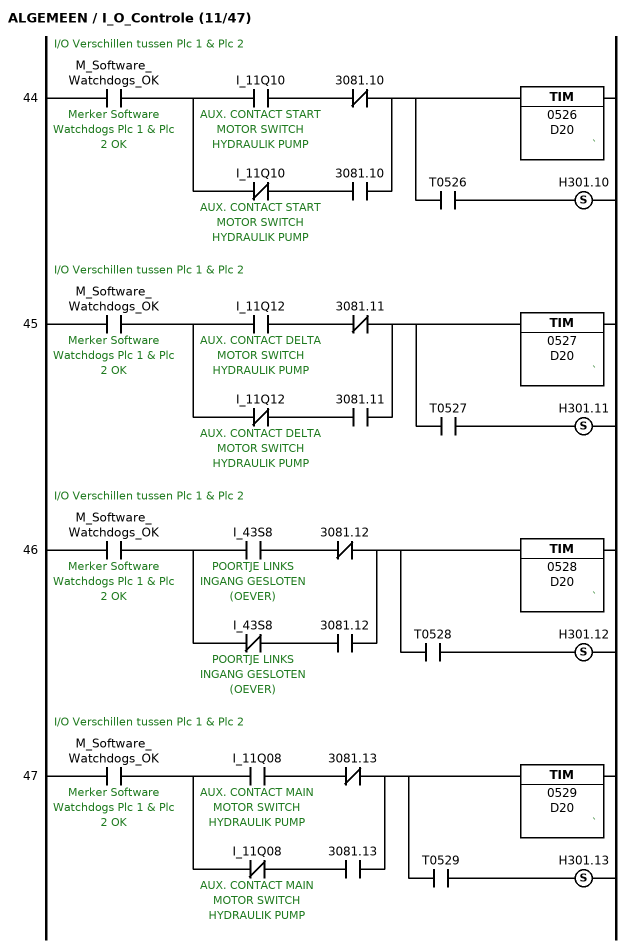
; rung 44: I/O Verschillen tussen Plc 1 & Plc 2
LD M_Software_Watchdogs_OK  ; Merker Software Watchdogs Plc 1 & Plc 2 OK
LD I_11Q10  ; AUX. CONTACT START MOTOR SWITCH HYDRAULIK PUMP
ANDNOT 3081.10
LDNOT I_11Q10  ; AUX. CONTACT START MOTOR SWITCH HYDRAULIK PUMP
AND 3081.10
ORLD
ANDLD
TIM 0526 D20  ; `
AND T0526
SET H301.10
; rung 45: I/O Verschillen tussen Plc 1 & Plc 2
LD M_Software_Watchdogs_OK  ; Merker Software Watchdogs Plc 1 & Plc 2 OK
LD I_11Q12  ; AUX. CONTACT DELTA MOTOR SWITCH HYDRAULIK PUMP
ANDNOT 3081.11
LDNOT I_11Q12  ; AUX. CONTACT DELTA MOTOR SWITCH HYDRAULIK PUMP
AND 3081.11
ORLD
ANDLD
TIM 0527 D20  ; `
AND T0527
SET H301.11
; rung 46: I/O Verschillen tussen Plc 1 & Plc 2
LD M_Software_Watchdogs_OK  ; Merker Software Watchdogs Plc 1 & Plc 2 OK
LD I_43S8  ; POORTJE LINKS INGANG GESLOTEN (OEVER)
ANDNOT 3081.12
LDNOT I_43S8  ; POORTJE LINKS INGANG GESLOTEN (OEVER)
AND 3081.12
ORLD
ANDLD
TIM 0528 D20  ; `
AND T0528
SET H301.12
; rung 47: I/O Verschillen tussen Plc 1 & Plc 2
LD M_Software_Watchdogs_OK  ; Merker Software Watchdogs Plc 1 & Plc 2 OK
LD I_11Q08  ; AUX. CONTACT MAIN MOTOR SWITCH HYDRAULIK PUMP
ANDNOT 3081.13
LDNOT I_11Q08  ; AUX. CONTACT MAIN MOTOR SWITCH HYDRAULIK PUMP
AND 3081.13
ORLD
ANDLD
TIM 0529 D20  ; `
AND T0529
SET H301.13

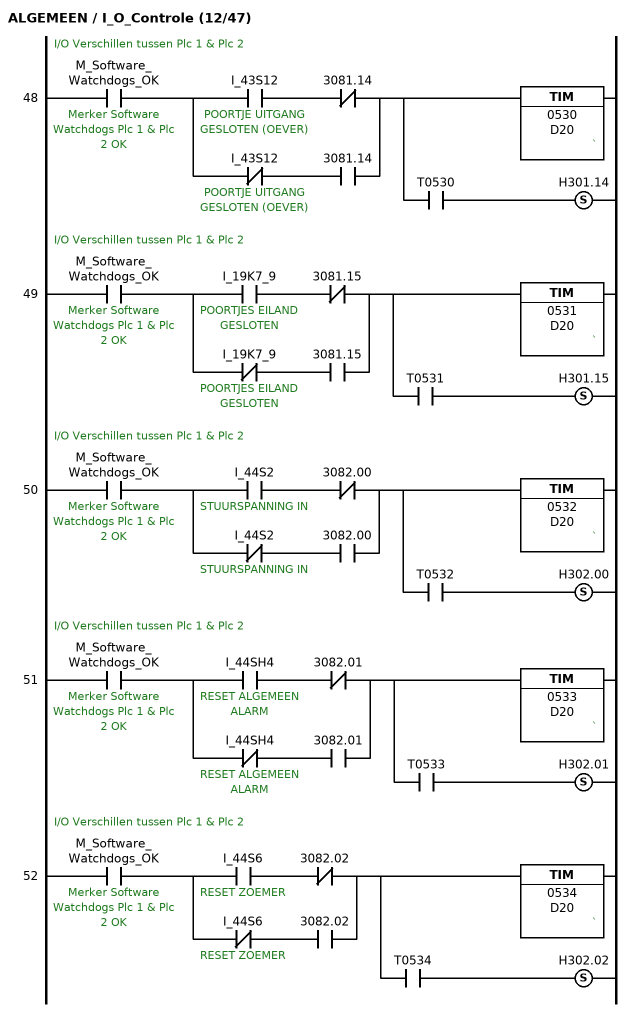
; rung 48: I/O Verschillen tussen Plc 1 & Plc 2
LD M_Software_Watchdogs_OK  ; Merker Software Watchdogs Plc 1 & Plc 2 OK
LD I_43S12  ; POORTJE UITGANG GESLOTEN (OEVER)
ANDNOT 3081.14
LDNOT I_43S12  ; POORTJE UITGANG GESLOTEN (OEVER)
AND 3081.14
ORLD
ANDLD
TIM 0530 D20  ; `
AND T0530
SET H301.14
; rung 49: I/O Verschillen tussen Plc 1 & Plc 2
LD M_Software_Watchdogs_OK  ; Merker Software Watchdogs Plc 1 & Plc 2 OK
LD I_19K7_9  ; POORTJES EILAND GESLOTEN
ANDNOT 3081.15
LDNOT I_19K7_9  ; POORTJES EILAND GESLOTEN
AND 3081.15
ORLD
ANDLD
TIM 0531 D20  ; `
AND T0531
SET H301.15
; rung 50: I/O Verschillen tussen Plc 1 & Plc 2
LD M_Software_Watchdogs_OK  ; Merker Software Watchdogs Plc 1 & Plc 2 OK
LD I_44S2  ; STUURSPANNING IN
ANDNOT 3082.00
LDNOT I_44S2  ; STUURSPANNING IN
AND 3082.00
ORLD
ANDLD
TIM 0532 D20  ; `
AND T0532
SET H302.00
; rung 51: I/O Verschillen tussen Plc 1 & Plc 2
LD M_Software_Watchdogs_OK  ; Merker Software Watchdogs Plc 1 & Plc 2 OK
LD I_44SH4  ; RESET ALGEMEEN ALARM
ANDNOT 3082.01
LDNOT I_44SH4  ; RESET ALGEMEEN ALARM
AND 3082.01
ORLD
ANDLD
TIM 0533 D20  ; `
AND T0533
SET H302.01
; rung 52: I/O Verschillen tussen Plc 1 & Plc 2
LD M_Software_Watchdogs_OK  ; Merker Software Watchdogs Plc 1 & Plc 2 OK
LD I_44S6  ; RESET ZOEMER
ANDNOT 3082.02
LDNOT I_44S6  ; RESET ZOEMER
AND 3082.02
ORLD
ANDLD
TIM 0534 D20  ; `
AND T0534
SET H302.02

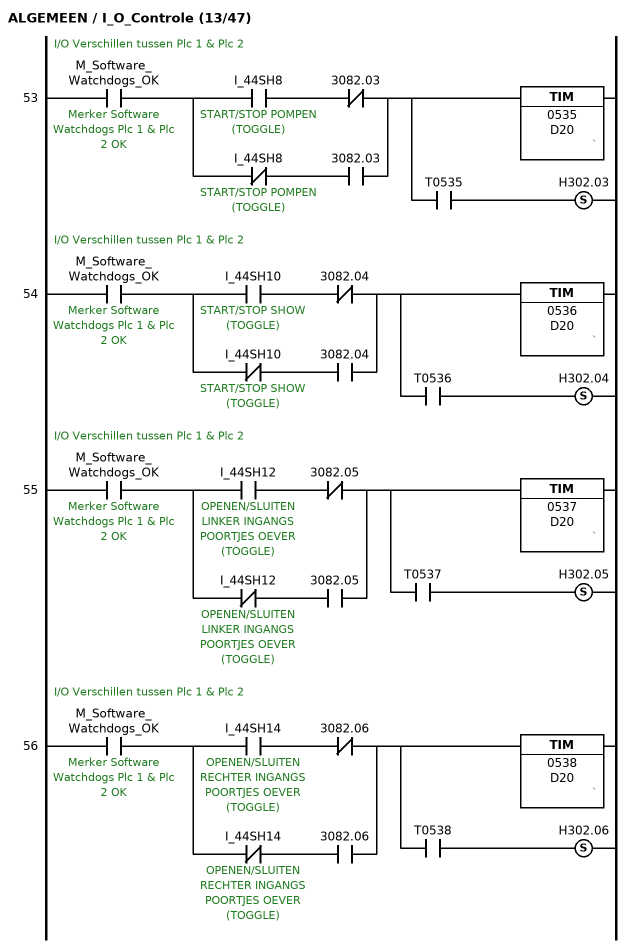
; rung 53: I/O Verschillen tussen Plc 1 & Plc 2
LD M_Software_Watchdogs_OK  ; Merker Software Watchdogs Plc 1 & Plc 2 OK
LD I_44SH8  ; START/STOP POMPEN (TOGGLE)
ANDNOT 3082.03
LDNOT I_44SH8  ; START/STOP POMPEN (TOGGLE)
AND 3082.03
ORLD
ANDLD
TIM 0535 D20  ; `
AND T0535
SET H302.03
; rung 54: I/O Verschillen tussen Plc 1 & Plc 2
LD M_Software_Watchdogs_OK  ; Merker Software Watchdogs Plc 1 & Plc 2 OK
LD I_44SH10  ; START/STOP SHOW (TOGGLE)
ANDNOT 3082.04
LDNOT I_44SH10  ; START/STOP SHOW (TOGGLE)
AND 3082.04
ORLD
ANDLD
TIM 0536 D20  ; `
AND T0536
SET H302.04
; rung 55: I/O Verschillen tussen Plc 1 & Plc 2
LD M_Software_Watchdogs_OK  ; Merker Software Watchdogs Plc 1 & Plc 2 OK
LD I_44SH12  ; OPENEN/SLUITEN LINKER INGANGS POORTJES OEVER  (TOGGLE)
ANDNOT 3082.05
LDNOT I_44SH12  ; OPENEN/SLUITEN LINKER INGANGS POORTJES OEVER  (TOGGLE)
AND 3082.05
ORLD
ANDLD
TIM 0537 D20  ; `
AND T0537
SET H302.05
; rung 56: I/O Verschillen tussen Plc 1 & Plc 2
LD M_Software_Watchdogs_OK  ; Merker Software Watchdogs Plc 1 & Plc 2 OK
LD I_44SH14  ; OPENEN/SLUITEN RECHTER INGANGS POORTJES OEVER  (TOGGLE)
ANDNOT 3082.06
LDNOT I_44SH14  ; OPENEN/SLUITEN RECHTER INGANGS POORTJES OEVER  (TOGGLE)
AND 3082.06
ORLD
ANDLD
TIM 0538 D20  ; `
AND T0538
SET H302.06

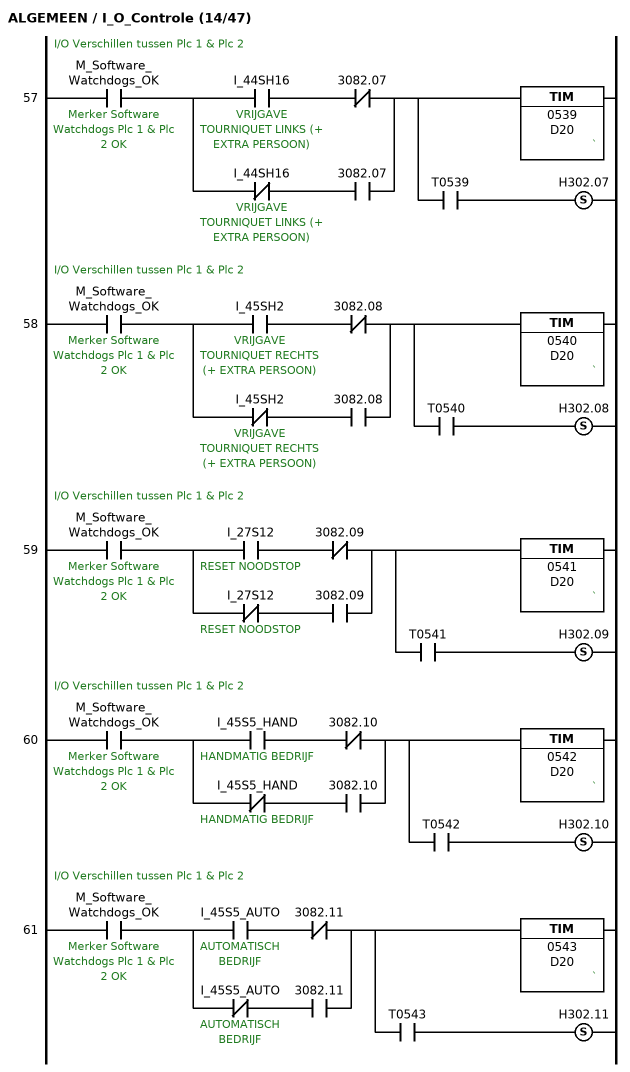
; rung 57: I/O Verschillen tussen Plc 1 & Plc 2
LD M_Software_Watchdogs_OK  ; Merker Software Watchdogs Plc 1 & Plc 2 OK
LD I_44SH16  ; VRIJGAVE TOURNIQUET LINKS (+ EXTRA PERSOON)
ANDNOT 3082.07
LDNOT I_44SH16  ; VRIJGAVE TOURNIQUET LINKS (+ EXTRA PERSOON)
AND 3082.07
ORLD
ANDLD
TIM 0539 D20  ; `
AND T0539
SET H302.07
; rung 58: I/O Verschillen tussen Plc 1 & Plc 2
LD M_Software_Watchdogs_OK  ; Merker Software Watchdogs Plc 1 & Plc 2 OK
LD I_45SH2  ; VRIJGAVE TOURNIQUET RECHTS (+ EXTRA PERSOON)
ANDNOT 3082.08
LDNOT I_45SH2  ; VRIJGAVE TOURNIQUET RECHTS (+ EXTRA PERSOON)
AND 3082.08
ORLD
ANDLD
TIM 0540 D20  ; `
AND T0540
SET H302.08
; rung 59: I/O Verschillen tussen Plc 1 & Plc 2
LD M_Software_Watchdogs_OK  ; Merker Software Watchdogs Plc 1 & Plc 2 OK
LD I_27S12  ; RESET NOODSTOP
ANDNOT 3082.09
LDNOT I_27S12  ; RESET NOODSTOP
AND 3082.09
ORLD
ANDLD
TIM 0541 D20  ; `
AND T0541
SET H302.09
; rung 60: I/O Verschillen tussen Plc 1 & Plc 2
LD M_Software_Watchdogs_OK  ; Merker Software Watchdogs Plc 1 & Plc 2 OK
LD I_45S5_HAND  ; HANDMATIG BEDRIJF
ANDNOT 3082.10
LDNOT I_45S5_HAND  ; HANDMATIG BEDRIJF
AND 3082.10
ORLD
ANDLD
TIM 0542 D20  ; `
AND T0542
SET H302.10
; rung 61: I/O Verschillen tussen Plc 1 & Plc 2
LD M_Software_Watchdogs_OK  ; Merker Software Watchdogs Plc 1 & Plc 2 OK
LD I_45S5_AUTO  ; AUTOMATISCH BEDRIJF
ANDNOT 3082.11
LDNOT I_45S5_AUTO  ; AUTOMATISCH BEDRIJF
AND 3082.11
ORLD
ANDLD
TIM 0543 D20  ; `
AND T0543
SET H302.11

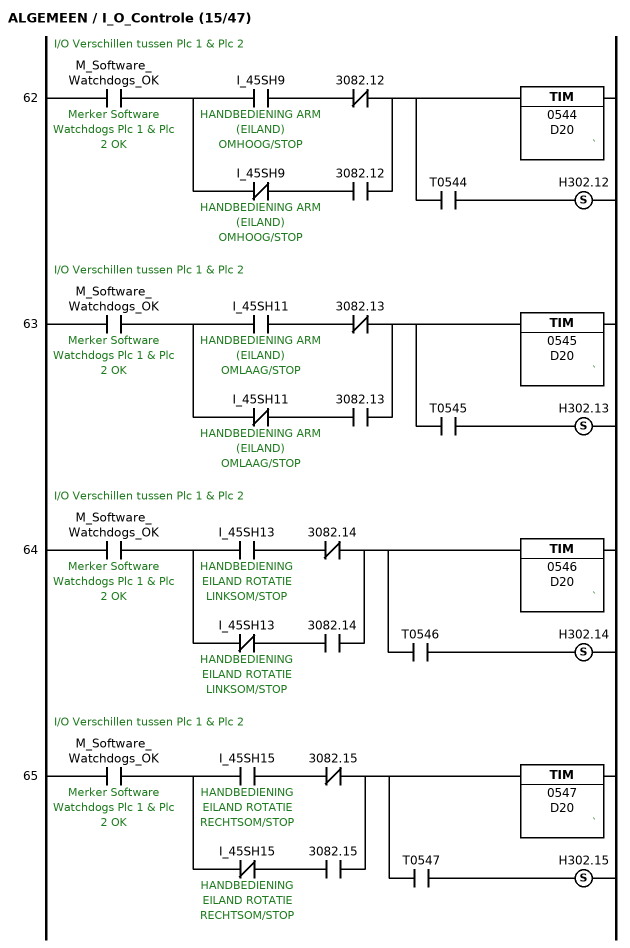
; rung 62: I/O Verschillen tussen Plc 1 & Plc 2
LD M_Software_Watchdogs_OK  ; Merker Software Watchdogs Plc 1 & Plc 2 OK
LD I_45SH9  ; HANDBEDIENING ARM (EILAND) OMHOOG/STOP
ANDNOT 3082.12
LDNOT I_45SH9  ; HANDBEDIENING ARM (EILAND) OMHOOG/STOP
AND 3082.12
ORLD
ANDLD
TIM 0544 D20  ; `
AND T0544
SET H302.12
; rung 63: I/O Verschillen tussen Plc 1 & Plc 2
LD M_Software_Watchdogs_OK  ; Merker Software Watchdogs Plc 1 & Plc 2 OK
LD I_45SH11  ; HANDBEDIENING ARM (EILAND) OMLAAG/STOP
ANDNOT 3082.13
LDNOT I_45SH11  ; HANDBEDIENING ARM (EILAND) OMLAAG/STOP
AND 3082.13
ORLD
ANDLD
TIM 0545 D20  ; `
AND T0545
SET H302.13
; rung 64: I/O Verschillen tussen Plc 1 & Plc 2
LD M_Software_Watchdogs_OK  ; Merker Software Watchdogs Plc 1 & Plc 2 OK
LD I_45SH13  ; HANDBEDIENING EILAND ROTATIE LINKSOM/STOP
ANDNOT 3082.14
LDNOT I_45SH13  ; HANDBEDIENING EILAND ROTATIE LINKSOM/STOP
AND 3082.14
ORLD
ANDLD
TIM 0546 D20  ; `
AND T0546
SET H302.14
; rung 65: I/O Verschillen tussen Plc 1 & Plc 2
LD M_Software_Watchdogs_OK  ; Merker Software Watchdogs Plc 1 & Plc 2 OK
LD I_45SH15  ; HANDBEDIENING EILAND ROTATIE RECHTSOM/STOP
ANDNOT 3082.15
LDNOT I_45SH15  ; HANDBEDIENING EILAND ROTATIE RECHTSOM/STOP
AND 3082.15
ORLD
ANDLD
TIM 0547 D20  ; `
AND T0547
SET H302.15

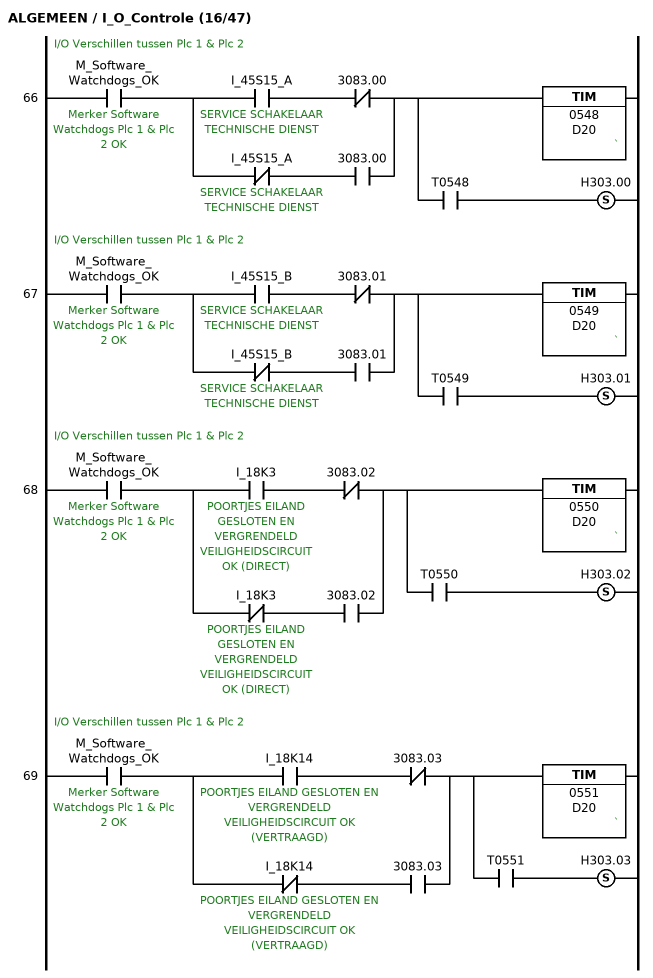
; rung 66: I/O Verschillen tussen Plc 1 & Plc 2
LD M_Software_Watchdogs_OK  ; Merker Software Watchdogs Plc 1 & Plc 2 OK
LD I_45S15_A  ; SERVICE SCHAKELAAR TECHNISCHE DIENST
ANDNOT 3083.00
LDNOT I_45S15_A  ; SERVICE SCHAKELAAR TECHNISCHE DIENST
AND 3083.00
ORLD
ANDLD
TIM 0548 D20  ; `
AND T0548
SET H303.00
; rung 67: I/O Verschillen tussen Plc 1 & Plc 2
LD M_Software_Watchdogs_OK  ; Merker Software Watchdogs Plc 1 & Plc 2 OK
LD I_45S15_B  ; SERVICE SCHAKELAAR TECHNISCHE DIENST
ANDNOT 3083.01
LDNOT I_45S15_B  ; SERVICE SCHAKELAAR TECHNISCHE DIENST
AND 3083.01
ORLD
ANDLD
TIM 0549 D20  ; `
AND T0549
SET H303.01
; rung 68: I/O Verschillen tussen Plc 1 & Plc 2
LD M_Software_Watchdogs_OK  ; Merker Software Watchdogs Plc 1 & Plc 2 OK
LD I_18K3  ; POORTJES EILAND GESLOTEN EN VERGRENDELD VEILIGHEIDSCIRCUIT OK (DIRECT)
ANDNOT 3083.02
LDNOT I_18K3  ; POORTJES EILAND GESLOTEN EN VERGRENDELD VEILIGHEIDSCIRCUIT OK (DIRECT)
AND 3083.02
ORLD
ANDLD
TIM 0550 D20  ; `
AND T0550
SET H303.02
; rung 69: I/O Verschillen tussen Plc 1 & Plc 2
LD M_Software_Watchdogs_OK  ; Merker Software Watchdogs Plc 1 & Plc 2 OK
LD I_18K14  ; POORTJES EILAND GESLOTEN EN VERGRENDELD VEILIGHEIDSCIRCUIT OK (VERTRAAGD)
ANDNOT 3083.03
LDNOT I_18K14  ; POORTJES EILAND GESLOTEN EN VERGRENDELD VEILIGHEIDSCIRCUIT OK (VERTRAAGD)
AND 3083.03
ORLD
ANDLD
TIM 0551 D20  ; `
AND T0551
SET H303.03

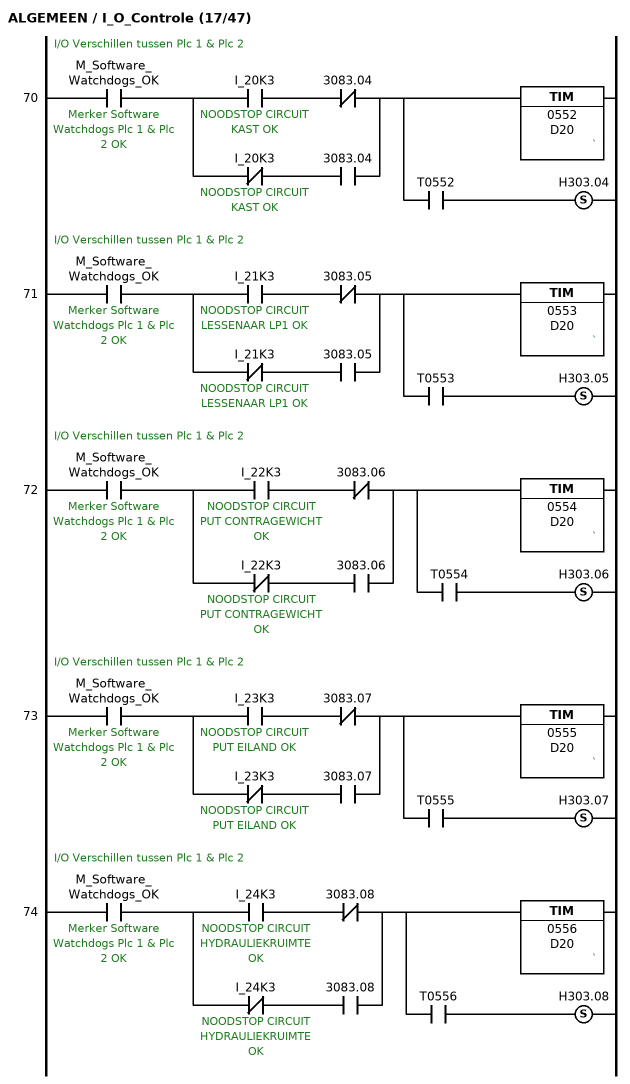
; rung 70: I/O Verschillen tussen Plc 1 & Plc 2
LD M_Software_Watchdogs_OK  ; Merker Software Watchdogs Plc 1 & Plc 2 OK
LD I_20K3  ; NOODSTOP CIRCUIT KAST OK
ANDNOT 3083.04
LDNOT I_20K3  ; NOODSTOP CIRCUIT KAST OK
AND 3083.04
ORLD
ANDLD
TIM 0552 D20  ; `
AND T0552
SET H303.04
; rung 71: I/O Verschillen tussen Plc 1 & Plc 2
LD M_Software_Watchdogs_OK  ; Merker Software Watchdogs Plc 1 & Plc 2 OK
LD I_21K3  ; NOODSTOP CIRCUIT LESSENAAR LP1 OK
ANDNOT 3083.05
LDNOT I_21K3  ; NOODSTOP CIRCUIT LESSENAAR LP1 OK
AND 3083.05
ORLD
ANDLD
TIM 0553 D20  ; `
AND T0553
SET H303.05
; rung 72: I/O Verschillen tussen Plc 1 & Plc 2
LD M_Software_Watchdogs_OK  ; Merker Software Watchdogs Plc 1 & Plc 2 OK
LD I_22K3  ; NOODSTOP CIRCUIT PUT CONTRAGEWICHT OK
ANDNOT 3083.06
LDNOT I_22K3  ; NOODSTOP CIRCUIT PUT CONTRAGEWICHT OK
AND 3083.06
ORLD
ANDLD
TIM 0554 D20  ; `
AND T0554
SET H303.06
; rung 73: I/O Verschillen tussen Plc 1 & Plc 2
LD M_Software_Watchdogs_OK  ; Merker Software Watchdogs Plc 1 & Plc 2 OK
LD I_23K3  ; NOODSTOP CIRCUIT PUT EILAND OK
ANDNOT 3083.07
LDNOT I_23K3  ; NOODSTOP CIRCUIT PUT EILAND OK
AND 3083.07
ORLD
ANDLD
TIM 0555 D20  ; `
AND T0555
SET H303.07
; rung 74: I/O Verschillen tussen Plc 1 & Plc 2
LD M_Software_Watchdogs_OK  ; Merker Software Watchdogs Plc 1 & Plc 2 OK
LD I_24K3  ; NOODSTOP CIRCUIT HYDRAULIEKRUIMTE OK
ANDNOT 3083.08
LDNOT I_24K3  ; NOODSTOP CIRCUIT HYDRAULIEKRUIMTE OK
AND 3083.08
ORLD
ANDLD
TIM 0556 D20  ; `
AND T0556
SET H303.08

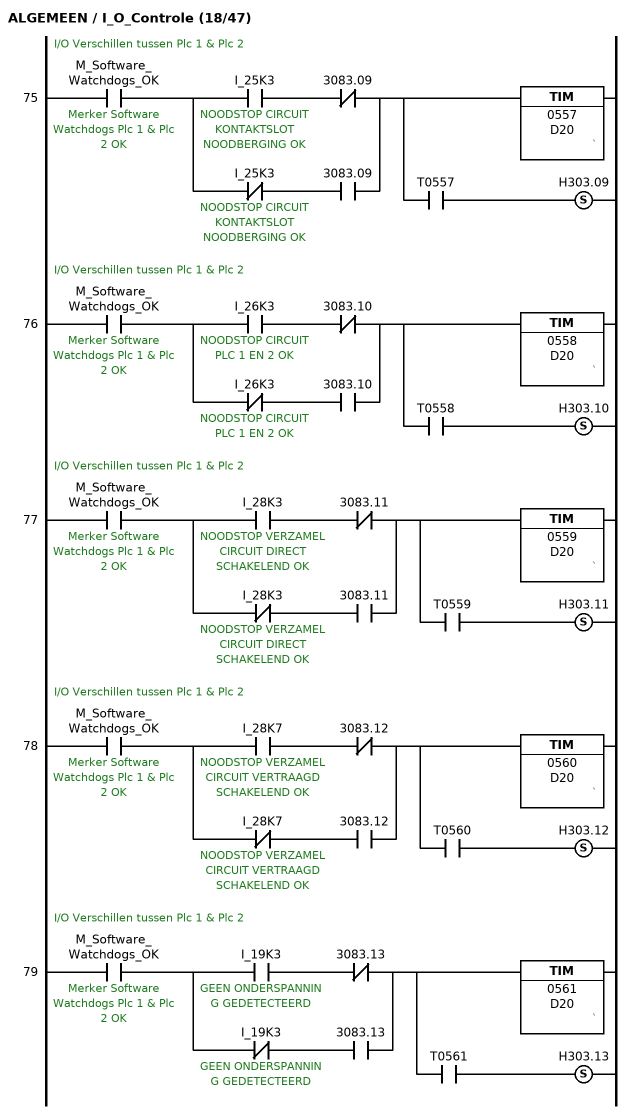
; rung 75: I/O Verschillen tussen Plc 1 & Plc 2
LD M_Software_Watchdogs_OK  ; Merker Software Watchdogs Plc 1 & Plc 2 OK
LD I_25K3  ; NOODSTOP CIRCUIT KONTAKTSLOT NOODBERGING OK
ANDNOT 3083.09
LDNOT I_25K3  ; NOODSTOP CIRCUIT KONTAKTSLOT NOODBERGING OK
AND 3083.09
ORLD
ANDLD
TIM 0557 D20  ; `
AND T0557
SET H303.09
; rung 76: I/O Verschillen tussen Plc 1 & Plc 2
LD M_Software_Watchdogs_OK  ; Merker Software Watchdogs Plc 1 & Plc 2 OK
LD I_26K3  ; NOODSTOP CIRCUIT PLC 1 EN 2 OK
ANDNOT 3083.10
LDNOT I_26K3  ; NOODSTOP CIRCUIT PLC 1 EN 2 OK
AND 3083.10
ORLD
ANDLD
TIM 0558 D20  ; `
AND T0558
SET H303.10
; rung 77: I/O Verschillen tussen Plc 1 & Plc 2
LD M_Software_Watchdogs_OK  ; Merker Software Watchdogs Plc 1 & Plc 2 OK
LD I_28K3  ; NOODSTOP VERZAMEL CIRCUIT DIRECT SCHAKELEND OK
ANDNOT 3083.11
LDNOT I_28K3  ; NOODSTOP VERZAMEL CIRCUIT DIRECT SCHAKELEND OK
AND 3083.11
ORLD
ANDLD
TIM 0559 D20  ; `
AND T0559
SET H303.11
; rung 78: I/O Verschillen tussen Plc 1 & Plc 2
LD M_Software_Watchdogs_OK  ; Merker Software Watchdogs Plc 1 & Plc 2 OK
LD I_28K7  ; NOODSTOP VERZAMEL CIRCUIT VERTRAAGD SCHAKELEND OK
ANDNOT 3083.12
LDNOT I_28K7  ; NOODSTOP VERZAMEL CIRCUIT VERTRAAGD SCHAKELEND OK
AND 3083.12
ORLD
ANDLD
TIM 0560 D20  ; `
AND T0560
SET H303.12
; rung 79: I/O Verschillen tussen Plc 1 & Plc 2
LD M_Software_Watchdogs_OK  ; Merker Software Watchdogs Plc 1 & Plc 2 OK
LD I_19K3  ; GEEN ONDERSPANNING GEDETECTEERD
ANDNOT 3083.13
LDNOT I_19K3  ; GEEN ONDERSPANNING GEDETECTEERD
AND 3083.13
ORLD
ANDLD
TIM 0561 D20  ; `
AND T0561
SET H303.13

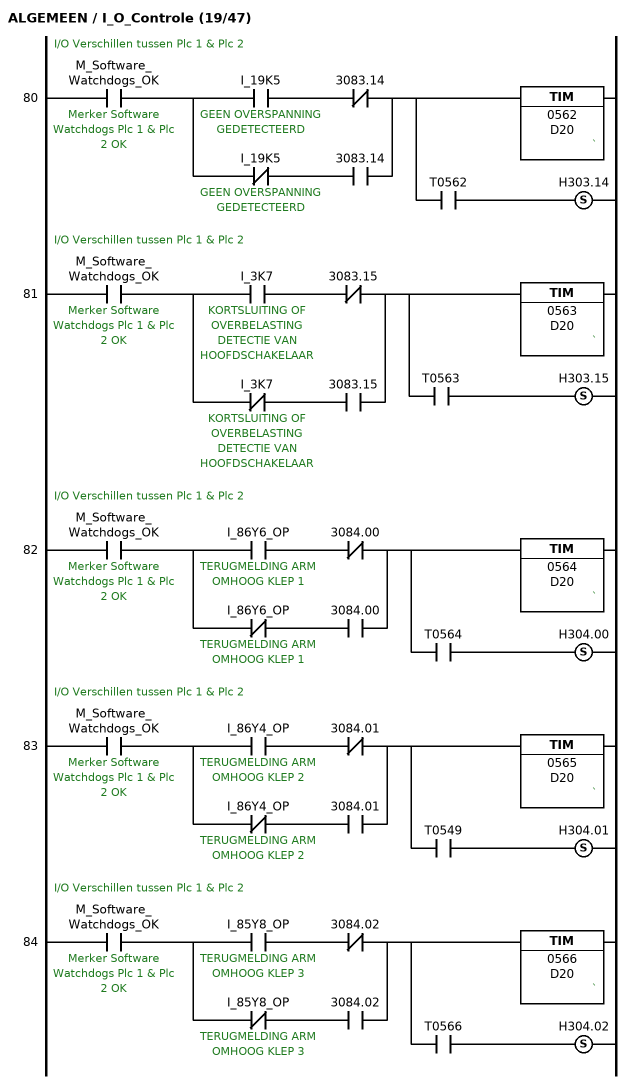
; rung 80: I/O Verschillen tussen Plc 1 & Plc 2
LD M_Software_Watchdogs_OK  ; Merker Software Watchdogs Plc 1 & Plc 2 OK
LD I_19K5  ; GEEN OVERSPANNING GEDETECTEERD
ANDNOT 3083.14
LDNOT I_19K5  ; GEEN OVERSPANNING GEDETECTEERD
AND 3083.14
ORLD
ANDLD
TIM 0562 D20  ; `
AND T0562
SET H303.14
; rung 81: I/O Verschillen tussen Plc 1 & Plc 2
LD M_Software_Watchdogs_OK  ; Merker Software Watchdogs Plc 1 & Plc 2 OK
LD I_3K7  ; KORTSLUITING OF OVERBELASTING DETECTIE VAN HOOFDSCHAKELAAR
ANDNOT 3083.15
LDNOT I_3K7  ; KORTSLUITING OF OVERBELASTING DETECTIE VAN HOOFDSCHAKELAAR
AND 3083.15
ORLD
ANDLD
TIM 0563 D20  ; `
AND T0563
SET H303.15
; rung 82: I/O Verschillen tussen Plc 1 & Plc 2
LD M_Software_Watchdogs_OK  ; Merker Software Watchdogs Plc 1 & Plc 2 OK
LD I_86Y6_OP  ; TERUGMELDING ARM OMHOOG KLEP 1
ANDNOT 3084.00
LDNOT I_86Y6_OP  ; TERUGMELDING ARM OMHOOG KLEP 1
AND 3084.00
ORLD
ANDLD
TIM 0564 D20  ; `
AND T0564
SET H304.00
; rung 83: I/O Verschillen tussen Plc 1 & Plc 2
LD M_Software_Watchdogs_OK  ; Merker Software Watchdogs Plc 1 & Plc 2 OK
LD I_86Y4_OP  ; TERUGMELDING ARM OMHOOG KLEP 2
ANDNOT 3084.01
LDNOT I_86Y4_OP  ; TERUGMELDING ARM OMHOOG KLEP 2
AND 3084.01
ORLD
ANDLD
TIM 0565 D20  ; `
AND T0549
SET H304.01
; rung 84: I/O Verschillen tussen Plc 1 & Plc 2
LD M_Software_Watchdogs_OK  ; Merker Software Watchdogs Plc 1 & Plc 2 OK
LD I_85Y8_OP  ; TERUGMELDING ARM OMHOOG KLEP 3
ANDNOT 3084.02
LDNOT I_85Y8_OP  ; TERUGMELDING ARM OMHOOG KLEP 3
AND 3084.02
ORLD
ANDLD
TIM 0566 D20  ; `
AND T0566
SET H304.02

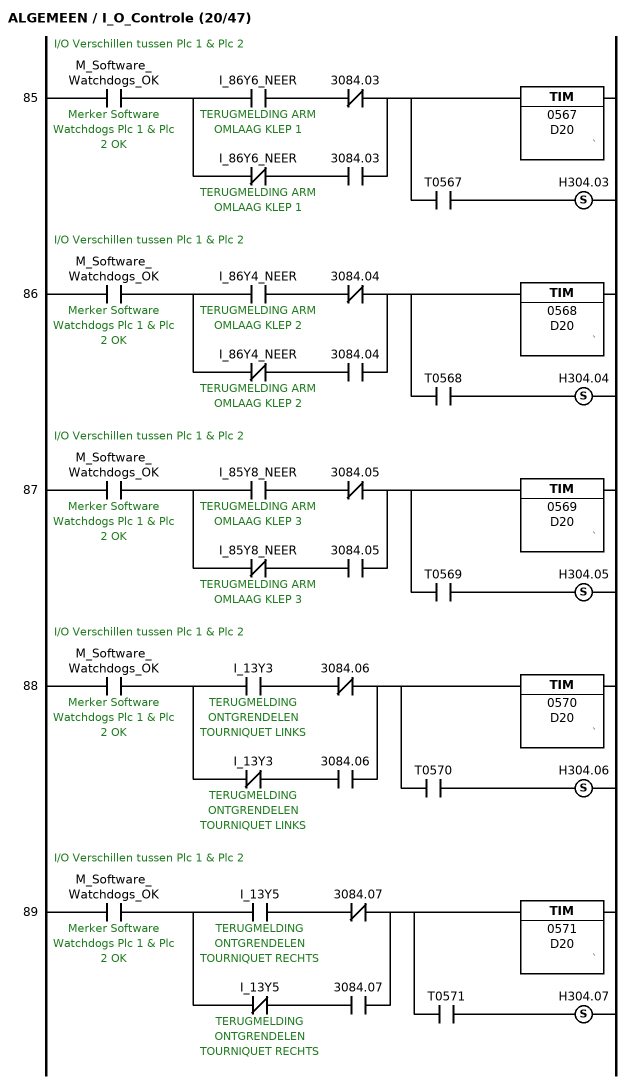
; rung 85: I/O Verschillen tussen Plc 1 & Plc 2
LD M_Software_Watchdogs_OK  ; Merker Software Watchdogs Plc 1 & Plc 2 OK
LD I_86Y6_NEER  ; TERUGMELDING ARM OMLAAG KLEP 1
ANDNOT 3084.03
LDNOT I_86Y6_NEER  ; TERUGMELDING ARM OMLAAG KLEP 1
AND 3084.03
ORLD
ANDLD
TIM 0567 D20  ; `
AND T0567
SET H304.03
; rung 86: I/O Verschillen tussen Plc 1 & Plc 2
LD M_Software_Watchdogs_OK  ; Merker Software Watchdogs Plc 1 & Plc 2 OK
LD I_86Y4_NEER  ; TERUGMELDING ARM OMLAAG KLEP 2
ANDNOT 3084.04
LDNOT I_86Y4_NEER  ; TERUGMELDING ARM OMLAAG KLEP 2
AND 3084.04
ORLD
ANDLD
TIM 0568 D20  ; `
AND T0568
SET H304.04
; rung 87: I/O Verschillen tussen Plc 1 & Plc 2
LD M_Software_Watchdogs_OK  ; Merker Software Watchdogs Plc 1 & Plc 2 OK
LD I_85Y8_NEER  ; TERUGMELDING ARM OMLAAG KLEP 3
ANDNOT 3084.05
LDNOT I_85Y8_NEER  ; TERUGMELDING ARM OMLAAG KLEP 3
AND 3084.05
ORLD
ANDLD
TIM 0569 D20  ; `
AND T0569
SET H304.05
; rung 88: I/O Verschillen tussen Plc 1 & Plc 2
LD M_Software_Watchdogs_OK  ; Merker Software Watchdogs Plc 1 & Plc 2 OK
LD I_13Y3  ; TERUGMELDING ONTGRENDELEN TOURNIQUET LINKS
ANDNOT 3084.06
LDNOT I_13Y3  ; TERUGMELDING ONTGRENDELEN TOURNIQUET LINKS
AND 3084.06
ORLD
ANDLD
TIM 0570 D20  ; `
AND T0570
SET H304.06
; rung 89: I/O Verschillen tussen Plc 1 & Plc 2
LD M_Software_Watchdogs_OK  ; Merker Software Watchdogs Plc 1 & Plc 2 OK
LD I_13Y5  ; TERUGMELDING ONTGRENDELEN TOURNIQUET RECHTS
ANDNOT 3084.07
LDNOT I_13Y5  ; TERUGMELDING ONTGRENDELEN TOURNIQUET RECHTS
AND 3084.07
ORLD
ANDLD
TIM 0571 D20  ; `
AND T0571
SET H304.07

